LIN {X 0,Y 474.677,Z 139.36,A -85,B 0,C 180,E1 -7395.457,E2 -7395.457} C_VEL
LIN {X 0,Y 474.649,Z 139.359,A -85,B 0,C 180,E1 -7399.011,E2 -7399.011} C_VEL
LIN {X 0,Y 474.578,Z 139.368,A -85,B 0,C 180,E1 -7401.73,E2 -7401.73} C_VEL
LIN {X 0,Y 474.616,Z 139.361,A -85,B 0,C 180,E1 -7404.495,E2 -7404.495} C_VEL
LIN {X 0,Y 474.629,Z 139.365,A -85,B 0,C 180,E1 -7407.325,E2 -7407.325} C_VEL
LIN {X 0,Y 474.588,Z 139.364,A -85,B 0,C 180,E1 -7410.232,E2 -7410.232} C_VEL
LIN {X 0,Y 474.607,Z 139.367,A -85,B 0,C 180,E1 -7413.223,E2 -7413.223} C_VEL
LIN {X 0,Y 474.581,Z 139.366,A -85,B 0,C 180,E1 -7416.324,E2 -7416.324} C_VEL
LIN {X 0,Y 474.615,Z 139.361,A -85,B 0,C 180,E1 -7419.549,E2 -7419.549} C_VEL
LIN {X 0,Y 474.578,Z 139.367,A -85,B 0,C 180,E1 -7422.232,E2 -7422.232} C_VEL
LIN {X 0,Y 474.611,Z 139.362,A -85,B 0,C 180,E1 -7425.299,E2 -7425.299} C_VEL
LIN {X 0,Y 474.61,Z 139.364,A -85,B 0,C 180,E1 -7428.215,E2 -7428.215} C_VEL
LIN {X 0,Y 474.605,Z 139.362,A -85,B 0,C 180,E1 -7431.543,E2 -7431.543} C_VEL
LIN {X 0,Y 474.619,Z 139.364,A -85,B 0,C 180,E1 -7434.726,E2 -7434.726} C_VEL
LIN {X 0,Y 474.633,Z 139.36,A -85,B 0,C 180,E1 -7437.789,E2 -7437.789} C_VEL
LIN {X 0,Y 474.597,Z 139.364,A -85,B 0,C 180,E1 -7440.891,E2 -7440.891} C_VEL
LIN {X 0,Y 474.609,Z 139.363,A -85,B 0,C 180,E1 -7443.626,E2 -7443.626} C_VEL
LIN {X 0,Y 474.634,Z 139.36,A -85,B 0,C 180,E1 -7446.643,E2 -7446.643} C_VEL
LIN {X 0,Y 474.709,Z 139.506,A -85,B 0,C 180,E1 -7449.301,E2 -7449.301} C_VEL
LIN {X 0,Y 475.543,Z 144.063,A -85,B 0,C 180,E1 -7450.291,E2 -7450.291} C_VEL
LIN {X 0,Y 475.076,Z 146.121,A -85,B 0,C 180,E1 -7450.692,E2 -7450.692} C_VEL
LIN {X 0,Y 472.301,Z 149.701,A -85,B 0,C 180,E1 -7451.293,E2 -7451.293} C_VEL
LIN {X 0,Y 469.325,Z 153.345,A -85,B 0,C 180,E1 -7451.896,E2 -7451.896} C_VEL
LIN {X 0,Y 468.584,Z 155.513,A -85,B 0,C 180,E1 -7452.3,E2 -7452.3} C_VEL
LIN {X 0,Y 468.493,Z 159.191,A -85,B 0,C 180,E1 -7453.033,E2 -7453.033} C_VEL
LIN {X 0,Y 471.458,Z 174.816,A -85,B 0,C 180,E1 -7453.399,E2 -7453.399} C_VEL
LIN {X 0,Y 470.697,Z 266.818,A -85,B 0,C 180,E1 -7454.826,E2 -7454.826} C_VEL
LIN {X 0,Y 470.413,Z 279.928,A -85,B 0,C 180,E1 -7455.204,E2 -7455.204} C_VEL
LIN {X 0,Y 470.036,Z 291.987,A -85,B 0,C 180,E1 -7455.718,E2 -7455.718} C_VEL
LIN {X 0,Y 469.631,Z 303.292,A -85,B 0,C 180,E1 -7456.364,E2 -7456.364} C_VEL
LIN {X 0,Y 469.304,Z 313.727,A -85,B 0,C 180,E1 -7457.13,E2 -7457.13} C_VEL
LIN {X 0,Y 468.722,Z 324.409,A -85,B 0,C 180,E1 -7458.103,E2 -7458.103} C_VEL
LIN {X 0,Y 468.281,Z 334.015,A -85,B 0,C 180,E1 -7459.188,E2 -7459.188} C_VEL
LIN {X 0,Y 467.829,Z 341.883,A -85,B 0,C 180,E1 -7460.271,E2 -7460.271} C_VEL
LIN {X 0,Y 467.434,Z 349.574,A -85,B 0,C 180,E1 -7461.571,E2 -7461.571} C_VEL
LIN {X 0,Y 467.127,Z 356.625,A -85,B 0,C 180,E1 -7463.088,E2 -7463.088} C_VEL
LIN {X 0,Y 466.942,Z 361.324,A -85,B 0,C 180,E1 -7464.386,E2 -7464.386} C_VEL
LIN {X 0,Y 466.844,Z 364.92,A -85,B 0,C 180,E1 -7465.684,E2 -7465.684} C_VEL
LIN {X 0,Y 466.817,Z 366.778,A -85,B 0,C 180,E1 -7466.548,E2 -7466.548} C_VEL
LIN {X 0,Y 466.718,Z 368.181,A -85,B 0,C 180,E1 -7467.411,E2 -7467.411} C_VEL
LIN {X 0,Y 466.626,Z 369.793,A -85,B 0,C 180,E1 -7469.137,E2 -7469.137} C_VEL
LIN {X 0,Y 466.607,Z 370.029,A -85,B 0,C 180,E1 -7470,E2 -7470} C_VEL
LIN {X 0,Y 466.626,Z 369.843,A -85,B 0,C 180,E1 -7470.863,E2 -7470.863} C_VEL
LIN {X 0,Y 466.719,Z 368.296,A -85,B 0,C 180,E1 -7472.59,E2 -7472.59} C_VEL
LIN {X 0,Y 466.818,Z 366.942,A -85,B 0,C 180,E1 -7473.453,E2 -7473.453} C_VEL
LIN {X 0,Y 466.819,Z 364.087,A -85,B 0,C 180,E1 -7474.75,E2 -7474.75} C_VEL
LIN {X 0,Y 467.063,Z 360.207,A -85,B 0,C 180,E1 -7476.047,E2 -7476.047} C_VEL
LIN {X 0,Y 467.173,Z 355.208,A -85,B 0,C 180,E1 -7477.347,E2 -7477.347} C_VEL
LIN {X 0,Y 467.498,Z 348.91,A -85,B 0,C 180,E1 -7478.647,E2 -7478.647} C_VEL
LIN {X 0,Y 467.886,Z 341.024,A -85,B 0,C 180,E1 -7479.947,E2 -7479.947} C_VEL
LIN {X 0,Y 468.262,Z 332.985,A -85,B 0,C 180,E1 -7481.032,E2 -7481.032} C_VEL
LIN {X 0,Y 468.813,Z 323.168,A -85,B 0,C 180,E1 -7482.115,E2 -7482.115} C_VEL
LIN {X 0,Y 469.318,Z 312.035,A -85,B 0,C 180,E1 -7483.099,E2 -7483.099} C_VEL
LIN {X 0,Y 469.813,Z 299.55,A -85,B 0,C 180,E1 -7483.959,E2 -7483.959} C_VEL
LIN {X 0,Y 470.211,Z 288.228,A -85,B 0,C 180,E1 -7484.554,E2 -7484.554} C_VEL
LIN {X 0,Y 470.55,Z 275.334,A -85,B 0,C 180,E1 -7485.041,E2 -7485.041} C_VEL
LIN {X 0,Y 470.828,Z 261.566,A -85,B 0,C 180,E1 -7485.364,E2 -7485.364} C_VEL
LIN {X 0,Y 471.336,Z 173.724,A -85,B 0,C 180,E1 -7486.716,E2 -7486.716} C_VEL
LIN {X 0,Y 468.504,Z 159.186,A -85,B 0,C 180,E1 -7487.061,E2 -7487.061} C_VEL
LIN {X 0,Y 468.83,Z 147.183,A -85,B 0,C 180,E1 -7489.484,E2 -7489.484} C_VEL
LIN {X 0,Y 467.636,Z 140.236,A -85,B 0,C 180,E1 -7491.027,E2 -7491.027} C_VEL
LIN {X 0,Y 467.559,Z 140.247,A -85,B 0,C 180,E1 -7493.944,E2 -7493.944} C_VEL
LIN {X 0,Y 467.564,Z 140.239,A -85,B 0,C 180,E1 -7496.804,E2 -7496.804} C_VEL
LIN {X 0,Y 467.548,Z 140.248,A -85,B 0,C 180,E1 -7499.739,E2 -7499.739} C_VEL
LIN {X 0,Y 467.585,Z 140.236,A -85,B 0,C 180,E1 -7502.758,E2 -7502.758} C_VEL
LIN {X 0,Y 467.552,Z 140.245,A -85,B 0,C 180,E1 -7505.89,E2 -7505.89} C_VEL
LIN {X 0,Y 467.553,Z 140.243,A -85,B 0,C 180,E1 -7509.148,E2 -7509.148} C_VEL
LIN {X 0,Y 467.567,Z 140.246,A -85,B 0,C 180,E1 -7511.404,E2 -7511.404} C_VEL
LIN {X 0,Y 467.565,Z 140.241,A -85,B 0,C 180,E1 -7514.947,E2 -7514.947} C_VEL
LIN {X 0,Y 467.56,Z 140.245,A -85,B 0,C 180,E1 -7517.436,E2 -7517.436} C_VEL
LIN {X 0,Y 467.563,Z 140.239,A -85,B 0,C 180,E1 -7520.048,E2 -7520.048} C_VEL
LIN {X 0,Y 467.522,Z 140.251,A -85,B 0,C 180,E1 -7523.037,E2 -7523.037} C_VEL
LIN {X 0,Y 467.565,Z 140.239,A -85,B 0,C 180,E1 -7526.21,E2 -7526.21} C_VEL
LIN {X 0,Y 467.561,Z 140.243,A -85,B 0,C 180,E1 -7529.265,E2 -7529.265} C_VEL
LIN {X 0,Y 467.573,Z 140.241,A -85,B 0,C 180,E1 -7532.475,E2 -7532.475} C_VEL
LIN {X 0,Y 467.566,Z 140.242,A -85,B 0,C 180,E1 -7535.11,E2 -7535.11} C_VEL
LIN {X 0,Y 467.531,Z 140.243,A -85,B 0,C 180,E1 -7537.926,E2 -7537.926} C_VEL
LIN {X 0,Y 467.615,Z 140.24,A -85,B 0,C 180,E1 -7540.692,E2 -7540.692} C_VEL
LIN {X 0,Y 467.609,Z 140.238,A -85,B 0,C 180,E1 -7544.304,E2 -7544.304} C_VEL
LIN {X 0,Y 467.653,Z 140.229,A -85,B 0,C 180,E1 -7547.854,E2 -7547.854} C_VEL
LIN {X 0,Y 467.653,Z 140.228,A -85,B 0,C 180,E1 -7551.357,E2 -7551.357} C_VEL
LIN {X 0,Y 467.696,Z 140.227,A -85,B 0,C 180,E1 -7553.962,E2 -7553.962} C_VEL
LIN {X 0,Y 467.808,Z 140.209,A -85,B 0,C 180,E1 -7557.417,E2 -7557.417} C_VEL
LIN {X 0,Y 467.845,Z 140.211,A -85,B 0,C 180,E1 -7560,E2 -7560} C_VEL
LIN {X 0,Y 467.806,Z 140.21,A -85,B 0,C 180,E1 -7562.583,E2 -7562.583} C_VEL
LIN {X 0,Y 467.695,Z 140.229,A -85,B 0,C 180,E1 -7566.038,E2 -7566.038} C_VEL
LIN {X 0,Y 467.625,Z 140.231,A -85,B 0,C 180,E1 -7568.644,E2 -7568.644} C_VEL
LIN {X 0,Y 467.637,Z 140.232,A -85,B 0,C 180,E1 -7572.146,E2 -7572.146} C_VEL
LIN {X 0,Y 467.573,Z 140.245,A -85,B 0,C 180,E1 -7575.697,E2 -7575.697} C_VEL
LIN {X 0,Y 467.568,Z 140.238,A -85,B 0,C 180,E1 -7578.748,E2 -7578.748} C_VEL
LIN {X 0,Y 467.555,Z 140.245,A -85,B 0,C 180,E1 -7581.261,E2 -7581.261} C_VEL
LIN {X 0,Y 467.545,Z 140.243,A -85,B 0,C 180,E1 -7583.945,E2 -7583.945} C_VEL
LIN {X 0,Y 467.531,Z 140.245,A -85,B 0,C 180,E1 -7586.806,E2 -7586.806} C_VEL
LIN {X 0,Y 467.507,Z 140.248,A -85,B 0,C 180,E1 -7589.742,E2 -7589.742} C_VEL
LIN {X 0,Y 467.57,Z 140.241,A -85,B 0,C 180,E1 -7592.76,E2 -7592.76} C_VEL
LIN {X 0,Y 467.547,Z 140.241,A -85,B 0,C 180,E1 -7595.89,E2 -7595.89} C_VEL
LIN {X 0,Y 467.55,Z 140.246,A -85,B 0,C 180,E1 -7599.148,E2 -7599.148} C_VEL
LIN {X 0,Y 467.557,Z 140.242,A -85,B 0,C 180,E1 -7601.405,E2 -7601.405} C_VEL
LIN {X 0,Y 467.564,Z 140.243,A -85,B 0,C 180,E1 -7605.053,E2 -7605.053} C_VEL
LIN {X 0,Y 467.56,Z 140.247,A -85,B 0,C 180,E1 -7608.726,E2 -7608.726} C_VEL
LIN {X 0,Y 467.561,Z 140.24,A -85,B 0,C 180,E1 -7611.955,E2 -7611.955} C_VEL
LIN {X 0,Y 467.556,Z 140.241,A -85,B 0,C 180,E1 -7615.167,E2 -7615.167} C_VEL
LIN {X 0,Y 467.579,Z 140.243,A -85,B 0,C 180,E1 -7618.26,E2 -7618.26} C_VEL
LIN {X 0,Y 467.546,Z 140.244,A -85,B 0,C 180,E1 -7621.248,E2 -7621.248} C_VEL
LIN {X 0,Y 467.617,Z 140.444,A -85,B 0,C 180,E1 -7623.981,E2 -7623.981} C_VEL
LIN {X 0,Y 469.837,Z 152.033,A -85,B 0,C 180,E1 -7626.179,E2 -7626.179} C_VEL
LIN {X 0,Y 469.312,Z 165.507,A -85,B 0,C 180,E1 -7628.541,E2 -7628.541} C_VEL
LIN {X 0,Y 468.516,Z 184.729,A -85,B 0,C 180,E1 -7631.865,E2 -7631.865} C_VEL
LIN {X 0,Y 468.292,Z 191.201,A -85,B 0,C 180,E1 -7632.976,E2 -7632.976} C_VEL
LIN {X 0,Y 471.193,Z 211.474,A -85,B 0,C 180,E1 -7633.399,E2 -7633.399} C_VEL
LIN {X 0,Y 470.529,Z 299.617,A -85,B 0,C 180,E1 -7634.764,E2 -7634.764} C_VEL
LIN {X 0,Y 470.159,Z 312.891,A -85,B 0,C 180,E1 -7635.14,E2 -7635.14} C_VEL
LIN {X 0,Y 469.717,Z 325.06,A -85,B 0,C 180,E1 -7635.652,E2 -7635.652} C_VEL
LIN {X 0,Y 469.181,Z 337.34,A -85,B 0,C 180,E1 -7636.354,E2 -7636.354} C_VEL
LIN {X 0,Y 468.645,Z 349.413,A -85,B 0,C 180,E1 -7637.26,E2 -7637.26} C_VEL
LIN {X 0,Y 468.147,Z 360.453,A -85,B 0,C 180,E1 -7638.307,E2 -7638.307} C_VEL
LIN {X 0,Y 467.678,Z 369.639,A -85,B 0,C 180,E1 -7639.392,E2 -7639.392} C_VEL
LIN {X 0,Y 467.26,Z 378.592,A -85,B 0,C 180,E1 -7640.695,E2 -7640.695} C_VEL
LIN {X 0,Y 466.993,Z 385.802,A -85,B 0,C 180,E1 -7641.998,E2 -7641.998} C_VEL
LIN {X 0,Y 466.831,Z 390.669,A -85,B 0,C 180,E1 -7643.082,E2 -7643.082} C_VEL
LIN {X 0,Y 466.73,Z 395.401,A -85,B 0,C 180,E1 -7644.383,E2 -7644.383} C_VEL
LIN {X 0,Y 466.646,Z 399.016,A -85,B 0,C 180,E1 -7645.681,E2 -7645.681} C_VEL
LIN {X 0,Y 466.689,Z 400.884,A -85,B 0,C 180,E1 -7646.546,E2 -7646.546} C_VEL
LIN {X 0,Y 466.662,Z 402.283,A -85,B 0,C 180,E1 -7647.41,E2 -7647.41} C_VEL
LIN {X 0,Y 466.623,Z 403.889,A -85,B 0,C 180,E1 -7649.137,E2 -7649.137} C_VEL
LIN {X 0,Y 466.605,Z 404.106,A -85,B 0,C 180,E1 -7650,E2 -7650} C_VEL
LIN {X 0,Y 466.623,Z 403.89,A -85,B 0,C 180,E1 -7650.863,E2 -7650.863} C_VEL
LIN {X 0,Y 466.662,Z 402.285,A -85,B 0,C 180,E1 -7652.589,E2 -7652.589} C_VEL
LIN {X 0,Y 466.689,Z 400.887,A -85,B 0,C 180,E1 -7653.453,E2 -7653.453} C_VEL
LIN {X 0,Y 466.687,Z 397.944,A -85,B 0,C 180,E1 -7654.751,E2 -7654.751} C_VEL
LIN {X 0,Y 466.741,Z 393.962,A -85,B 0,C 180,E1 -7656.05,E2 -7656.05} C_VEL
LIN {X 0,Y 466.938,Z 387.841,A -85,B 0,C 180,E1 -7657.567,E2 -7657.567} C_VEL
LIN {X 0,Y 467.157,Z 381.152,A -85,B 0,C 180,E1 -7658.87,E2 -7658.87} C_VEL
LIN {X 0,Y 467.512,Z 372.856,A -85,B 0,C 180,E1 -7660.173,E2 -7660.173} C_VEL
LIN {X 0,Y 467.972,Z 364.359,A -85,B 0,C 180,E1 -7661.258,E2 -7661.258} C_VEL
LIN {X 0,Y 468.448,Z 354.322,A -85,B 0,C 180,E1 -7662.301,E2 -7662.301} C_VEL
LIN {X 0,Y 468.93,Z 343.472,A -85,B 0,C 180,E1 -7663.211,E2 -7663.211} C_VEL
LIN {X 0,Y 469.421,Z 332.089,A -85,B 0,C 180,E1 -7663.97,E2 -7663.97} C_VEL
LIN {X 0,Y 469.874,Z 320.415,A -85,B 0,C 180,E1 -7664.564,E2 -7664.564} C_VEL
LIN {X 0,Y 470.37,Z 306.969,A -85,B 0,C 180,E1 -7665.046,E2 -7665.046} C_VEL
LIN {X 0,Y 470.624,Z 293.68,A -85,B 0,C 180,E1 -7665.343,E2 -7665.343} C_VEL
LIN {X 0,Y 471.058,Z 209.349,A -85,B 0,C 180,E1 -7666.637,E2 -7666.637} C_VEL
LIN {X 0,Y 468.285,Z 191.129,A -85,B 0,C 180,E1 -7667.034,E2 -7667.034} C_VEL
LIN {X 0,Y 468.906,Z 174.273,A -85,B 0,C 180,E1 -7669.936,E2 -7669.936} C_VEL
LIN {X 0,Y 469.661,Z 157.261,A -85,B 0,C 180,E1 -7672.895,E2 -7672.895} C_VEL
LIN {X 0,Y 469.837,Z 152.015,A -85,B 0,C 180,E1 -7673.82,E2 -7673.82} C_VEL
LIN {X 0,Y 467.571,Z 140.245,A -85,B 0,C 180,E1 -7676.081,E2 -7676.081} C_VEL
LIN {X 0,Y 467.548,Z 140.247,A -85,B 0,C 180,E1 -7679.327,E2 -7679.327} C_VEL
LIN {X 0,Y 467.575,Z 140.243,A -85,B 0,C 180,E1 -7681.74,E2 -7681.74} C_VEL
LIN {X 0,Y 467.552,Z 140.241,A -85,B 0,C 180,E1 -7684.833,E2 -7684.833} C_VEL
LIN {X 0,Y 467.557,Z 140.241,A -85,B 0,C 180,E1 -7688.044,E2 -7688.044} C_VEL
LIN {X 0,Y 467.559,Z 140.246,A -85,B 0,C 180,E1 -7691.403,E2 -7691.403} C_VEL
LIN {X 0,Y 467.559,Z 140.245,A -85,B 0,C 180,E1 -7695.052,E2 -7695.052} C_VEL
LIN {X 0,Y 467.554,Z 140.243,A -85,B 0,C 180,E1 -7698.725,E2 -7698.725} C_VEL
LIN {X 0,Y 467.554,Z 140.24,A -85,B 0,C 180,E1 -7701.954,E2 -7701.954} C_VEL
LIN {X 0,Y 467.548,Z 140.246,A -85,B 0,C 180,E1 -7705.166,E2 -7705.166} C_VEL
LIN {X 0,Y 467.549,Z 140.242,A -85,B 0,C 180,E1 -7708.257,E2 -7708.257} C_VEL
LIN {X 0,Y 467.535,Z 140.245,A -85,B 0,C 180,E1 -7711.248,E2 -7711.248} C_VEL
LIN {X 0,Y 467.568,Z 140.243,A -85,B 0,C 180,E1 -7714.4,E2 -7714.4} C_VEL
LIN {X 0,Y 467.559,Z 140.242,A -85,B 0,C 180,E1 -7716.995,E2 -7716.995} C_VEL
LIN {X 0,Y 467.6,Z 140.235,A -85,B 0,C 180,E1 -7719.776,E2 -7719.776} C_VEL
LIN {X 0,Y 467.551,Z 140.248,A -85,B 0,C 180,E1 -7722.505,E2 -7722.505} C_VEL
LIN {X 0,Y 467.58,Z 140.237,A -85,B 0,C 180,E1 -7725.196,E2 -7725.196} C_VEL
LIN {X 0,Y 467.637,Z 140.232,A -85,B 0,C 180,E1 -7727.854,E2 -7727.854} C_VEL
LIN {X 0,Y 467.622,Z 140.232,A -85,B 0,C 180,E1 -7731.356,E2 -7731.356} C_VEL
LIN {X 0,Y 467.689,Z 140.229,A -85,B 0,C 180,E1 -7733.962,E2 -7733.962} C_VEL
LIN {X 0,Y 467.8,Z 140.21,A -85,B 0,C 180,E1 -7737.417,E2 -7737.417} C_VEL
LIN {X 0,Y 467.838,Z 140.212,A -85,B 0,C 180,E1 -7740,E2 -7740} C_VEL
LIN {X 0,Y 467.802,Z 140.21,A -85,B 0,C 180,E1 -7742.583,E2 -7742.583} C_VEL
LIN {X 0,Y 467.693,Z 140.227,A -85,B 0,C 180,E1 -7746.038,E2 -7746.038} C_VEL
LIN {X 0,Y 467.656,Z 140.227,A -85,B 0,C 180,E1 -7748.643,E2 -7748.643} C_VEL
LIN {X 0,Y 467.646,Z 140.23,A -85,B 0,C 180,E1 -7752.146,E2 -7752.146} C_VEL
LIN {X 0,Y 467.602,Z 140.24,A -85,B 0,C 180,E1 -7755.696,E2 -7755.696} C_VEL
LIN {X 0,Y 467.609,Z 140.24,A -85,B 0,C 180,E1 -7759.308,E2 -7759.308} C_VEL
LIN {X 0,Y 467.521,Z 140.245,A -85,B 0,C 180,E1 -7762.075,E2 -7762.075} C_VEL
LIN {X 0,Y 467.55,Z 140.244,A -85,B 0,C 180,E1 -7764.891,E2 -7764.891} C_VEL
LIN {X 0,Y 467.552,Z 140.242,A -85,B 0,C 180,E1 -7767.774,E2 -7767.774} C_VEL
LIN {X 0,Y 467.557,Z 140.247,A -85,B 0,C 180,E1 -7771.045,E2 -7771.045} C_VEL
LIN {X 0,Y 467.569,Z 140.238,A -85,B 0,C 180,E1 -7774.241,E2 -7774.241} C_VEL
LIN {X 0,Y 467.54,Z 140.246,A -85,B 0,C 180,E1 -7777.187,E2 -7777.187} C_VEL
LIN {X 0,Y 467.551,Z 140.242,A -85,B 0,C 180,E1 -7780.268,E2 -7780.268} C_VEL
LIN {X 0,Y 467.54,Z 140.242,A -85,B 0,C 180,E1 -7783.747,E2 -7783.747} C_VEL
LIN {X 0,Y 467.544,Z 140.244,A -85,B 0,C 180,E1 -7786.256,E2 -7786.256} C_VEL
LIN {X 0,Y 467.565,Z 140.239,A -85,B 0,C 180,E1 -7789.735,E2 -7789.735} C_VEL
LIN {X 0,Y 467.539,Z 140.246,A -85,B 0,C 180,E1 -7792.816,E2 -7792.816} C_VEL
LIN {X 0,Y 467.584,Z 140.242,A -85,B 0,C 180,E1 -7796.213,E2 -7796.213} C_VEL
LIN {X 0,Y 467.564,Z 140.239,A -85,B 0,C 180,E1 -7799.267,E2 -7799.267} C_VEL
LIN {X 0,Y 467.573,Z 140.242,A -85,B 0,C 180,E1 -7802.476,E2 -7802.476} C_VEL
LIN {X 0,Y 467.567,Z 140.238,A -85,B 0,C 180,E1 -7805.112,E2 -7805.112} C_VEL
LIN {X 0,Y 467.534,Z 140.249,A -85,B 0,C 180,E1 -7807.927,E2 -7807.927} C_VEL
LIN {X 0,Y 467.639,Z 140.342,A -85,B 0,C 180,E1 -7809.118,E2 -7809.118} C_VEL
LIN {X 0,Y 468.8,Z 146.733,A -85,B 0,C 180,E1 -7810.516,E2 -7810.516} C_VEL
LIN {X 0,Y 468.584,Z 155.513,A -85,B 0,C 180,E1 -7812.3,E2 -7812.3} C_VEL
LIN {X 0,Y 468.186,Z 157.697,A -85,B 0,C 180,E1 -7812.596,E2 -7812.596} C_VEL
LIN {X 0,Y 467.029,Z 161.3,A -85,B 0,C 180,E1 -7812.843,E2 -7812.843} C_VEL
LIN {X 0,Y 465.264,Z 166.866,A -85,B 0,C 180,E1 -7813.019,E2 -7813.019} C_VEL
LIN {X 0,Y 464.706,Z 170.912,A -85,B 0,C 180,E1 -7813.084,E2 -7813.084} C_VEL
LIN {X 0,Y 465.202,Z 178.355,A -85,B 0,C 180,E1 -7813.219,E2 -7813.219} C_VEL
LIN {X 0,Y 464.513,Z 185.835,A -85,B 0,C 180,E1 -7813.313,E2 -7813.313} C_VEL
LIN {X 0,Y 463.852,Z 267.095,A -85,B 0,C 180,E1 -7814.597,E2 -7814.597} C_VEL
LIN {X 0,Y 463.565,Z 280.958,A -85,B 0,C 180,E1 -7815.009,E2 -7815.009} C_VEL
LIN {X 0,Y 463.147,Z 293.361,A -85,B 0,C 180,E1 -7815.557,E2 -7815.557} C_VEL
LIN {X 0,Y 462.704,Z 305.342,A -85,B 0,C 180,E1 -7816.281,E2 -7816.281} C_VEL
LIN {X 0,Y 462.305,Z 316.561,A -85,B 0,C 180,E1 -7817.155,E2 -7817.155} C_VEL
LIN {X 0,Y 461.692,Z 326.795,A -85,B 0,C 180,E1 -7818.142,E2 -7818.142} C_VEL
LIN {X 0,Y 461.227,Z 335.973,A -85,B 0,C 180,E1 -7819.243,E2 -7819.243} C_VEL
LIN {X 0,Y 460.729,Z 344.88,A -85,B 0,C 180,E1 -7820.563,E2 -7820.563} C_VEL
LIN {X 0,Y 460.301,Z 352.051,A -85,B 0,C 180,E1 -7821.881,E2 -7821.881} C_VEL
LIN {X 0,Y 460.058,Z 357.769,A -85,B 0,C 180,E1 -7823.2,E2 -7823.2} C_VEL
LIN {X 0,Y 459.899,Z 361.583,A -85,B 0,C 180,E1 -7824.3,E2 -7824.3} C_VEL
LIN {X 0,Y 459.752,Z 365.181,A -85,B 0,C 180,E1 -7825.617,E2 -7825.617} C_VEL
LIN {X 0,Y 459.75,Z 367.037,A -85,B 0,C 180,E1 -7826.495,E2 -7826.495} C_VEL
LIN {X 0,Y 459.641,Z 368.441,A -85,B 0,C 180,E1 -7827.371,E2 -7827.371} C_VEL
LIN {X 0,Y 459.559,Z 370.052,A -85,B 0,C 180,E1 -7829.124,E2 -7829.124} C_VEL
LIN {X 0,Y 459.538,Z 370.287,A -85,B 0,C 180,E1 -7830,E2 -7830} C_VEL
LIN {X 0,Y 459.559,Z 370.101,A -85,B 0,C 180,E1 -7830.877,E2 -7830.877} C_VEL
LIN {X 0,Y 459.641,Z 368.554,A -85,B 0,C 180,E1 -7832.63,E2 -7832.63} C_VEL
LIN {X 0,Y 459.75,Z 367.199,A -85,B 0,C 180,E1 -7833.506,E2 -7833.506} C_VEL
LIN {X 0,Y 459.735,Z 364.345,A -85,B 0,C 180,E1 -7834.823,E2 -7834.823} C_VEL
LIN {X 0,Y 460.01,Z 360.464,A -85,B 0,C 180,E1 -7836.14,E2 -7836.14} C_VEL
LIN {X 0,Y 460.129,Z 355.465,A -85,B 0,C 180,E1 -7837.46,E2 -7837.46} C_VEL
LIN {X 0,Y 460.48,Z 349.167,A -85,B 0,C 180,E1 -7838.779,E2 -7838.779} C_VEL
LIN {X 0,Y 460.88,Z 341.281,A -85,B 0,C 180,E1 -7840.1,E2 -7840.1} C_VEL
LIN {X 0,Y 461.305,Z 333.24,A -85,B 0,C 180,E1 -7841.201,E2 -7841.201} C_VEL
LIN {X 0,Y 461.897,Z 323.422,A -85,B 0,C 180,E1 -7842.299,E2 -7842.299} C_VEL
LIN {X 0,Y 462.394,Z 312.863,A -85,B 0,C 180,E1 -7843.253,E2 -7843.253} C_VEL
LIN {X 0,Y 462.873,Z 301.561,A -85,B 0,C 180,E1 -7844.06,E2 -7844.06} C_VEL
LIN {X 0,Y 463.348,Z 289.604,A -85,B 0,C 180,E1 -7844.718,E2 -7844.718} C_VEL
LIN {X 0,Y 463.702,Z 276.492,A -85,B 0,C 180,E1 -7845.24,E2 -7845.24} C_VEL
LIN {X 0,Y 463.973,Z 263.305,A -85,B 0,C 180,E1 -7845.569,E2 -7845.569} C_VEL
LIN {X 0,Y 464.537,Z 174.717,A -85,B 0,C 180,E1 -7846.956,E2 -7846.956} C_VEL
LIN {X 0,Y 461.559,Z 159.464,A -85,B 0,C 180,E1 -7847.319,E2 -7847.319} C_VEL
LIN {X 0,Y 461.891,Z 148.48,A -85,B 0,C 180,E1 -7849.557,E2 -7849.557} C_VEL
LIN {X 0,Y 460.55,Z 141.119,A -85,B 0,C 180,E1 -7851.218,E2 -7851.218} C_VEL
LIN {X 0,Y 460.524,Z 141.12,A -85,B 0,C 180,E1 -7854.333,E2 -7854.333} C_VEL
LIN {X 0,Y 460.535,Z 141.115,A -85,B 0,C 180,E1 -7857.246,E2 -7857.246} C_VEL
LIN {X 0,Y 460.508,Z 141.12,A -85,B 0,C 180,E1 -7860.24,E2 -7860.24} C_VEL
LIN {X 0,Y 460.531,Z 141.118,A -85,B 0,C 180,E1 -7863.325,E2 -7863.325} C_VEL
LIN {X 0,Y 460.474,Z 141.122,A -85,B 0,C 180,E1 -7866.53,E2 -7866.53} C_VEL
LIN {X 0,Y 460.514,Z 141.12,A -85,B 0,C 180,E1 -7869.864,E2 -7869.864} C_VEL
LIN {X 0,Y 460.493,Z 141.121,A -85,B 0,C 180,E1 -7872.897,E2 -7872.897} C_VEL
LIN {X 0,Y 460.505,Z 141.12,A -85,B 0,C 180,E1 -7875.831,E2 -7875.831} C_VEL
LIN {X 0,Y 460.519,Z 141.121,A -85,B 0,C 180,E1 -7878.987,E2 -7878.987} C_VEL
LIN {X 0,Y 460.513,Z 141.124,A -85,B 0,C 180,E1 -7881.265,E2 -7881.265} C_VEL
LIN {X 0,Y 460.505,Z 141.12,A -85,B 0,C 180,E1 -7884.554,E2 -7884.554} C_VEL
LIN {X 0,Y 460.516,Z 141.117,A -85,B 0,C 180,E1 -7887.714,E2 -7887.714} C_VEL
LIN {X 0,Y 460.518,Z 141.123,A -85,B 0,C 180,E1 -7890.767,E2 -7890.767} C_VEL
LIN {X 0,Y 460.527,Z 141.115,A -85,B 0,C 180,E1 -7893.732,E2 -7893.732} C_VEL
LIN {X 0,Y 460.541,Z 141.12,A -85,B 0,C 180,E1 -7896.624,E2 -7896.624} C_VEL
LIN {X 0,Y 460.546,Z 141.113,A -85,B 0,C 180,E1 -7899.452,E2 -7899.452} C_VEL
LIN {X 0,Y 460.521,Z 141.119,A -85,B 0,C 180,E1 -7902.229,E2 -7902.229} C_VEL
LIN {X 0,Y 460.545,Z 141.116,A -85,B 0,C 180,E1 -7904.964,E2 -7904.964} C_VEL
LIN {X 0,Y 460.605,Z 141.111,A -85,B 0,C 180,E1 -7908.559,E2 -7908.559} C_VEL
LIN {X 0,Y 460.605,Z 141.106,A -85,B 0,C 180,E1 -7911.223,E2 -7911.223} C_VEL
LIN {X 0,Y 460.662,Z 141.102,A -85,B 0,C 180,E1 -7913.869,E2 -7913.869} C_VEL
LIN {X 0,Y 460.752,Z 141.088,A -85,B 0,C 180,E1 -7917.377,E2 -7917.377} C_VEL
LIN {X 0,Y 460.814,Z 141.087,A -85,B 0,C 180,E1 -7920,E2 -7920} C_VEL
LIN {X 0,Y 460.75,Z 141.089,A -85,B 0,C 180,E1 -7922.623,E2 -7922.623} C_VEL
LIN {X 0,Y 460.661,Z 141.104,A -85,B 0,C 180,E1 -7926.131,E2 -7926.131} C_VEL
LIN {X 0,Y 460.58,Z 141.109,A -85,B 0,C 180,E1 -7928.777,E2 -7928.777} C_VEL
LIN {X 0,Y 460.594,Z 141.108,A -85,B 0,C 180,E1 -7932.435,E2 -7932.435} C_VEL
LIN {X 0,Y 460.522,Z 141.119,A -85,B 0,C 180,E1 -7935.965,E2 -7935.965} C_VEL
LIN {X 0,Y 460.527,Z 141.116,A -85,B 0,C 180,E1 -7938.886,E2 -7938.886} C_VEL
LIN {X 0,Y 460.506,Z 141.126,A -85,B 0,C 180,E1 -7941.486,E2 -7941.486} C_VEL
LIN {X 0,Y 460.51,Z 141.117,A -85,B 0,C 180,E1 -7944.334,E2 -7944.334} C_VEL
LIN {X 0,Y 460.486,Z 141.128,A -85,B 0,C 180,E1 -7947.249,E2 -7947.249} C_VEL
LIN {X 0,Y 460.476,Z 141.122,A -85,B 0,C 180,E1 -7950.243,E2 -7950.243} C_VEL
LIN {X 0,Y 460.513,Z 141.122,A -85,B 0,C 180,E1 -7953.326,E2 -7953.326} C_VEL
LIN {X 0,Y 460.469,Z 141.125,A -85,B 0,C 180,E1 -7956.53,E2 -7956.53} C_VEL
LIN {X 0,Y 460.511,Z 141.117,A -85,B 0,C 180,E1 -7959.865,E2 -7959.865} C_VEL
LIN {X 0,Y 460.461,Z 141.131,A -85,B 0,C 180,E1 -7962.894,E2 -7962.894} C_VEL
LIN {X 0,Y 460.502,Z 141.118,A -85,B 0,C 180,E1 -7965.832,E2 -7965.832} C_VEL
LIN {X 0,Y 460.514,Z 141.121,A -85,B 0,C 180,E1 -7968.987,E2 -7968.987} C_VEL
LIN {X 0,Y 460.498,Z 141.124,A -85,B 0,C 180,E1 -7972.377,E2 -7972.377} C_VEL
LIN {X 0,Y 460.536,Z 141.114,A -85,B 0,C 180,E1 -7975.623,E2 -7975.623} C_VEL
LIN {X 0,Y 460.539,Z 141.119,A -85,B 0,C 180,E1 -7978.745,E2 -7978.745} C_VEL
LIN {X 0,Y 460.533,Z 141.122,A -85,B 0,C 180,E1 -7982.266,E2 -7982.266} C_VEL
LIN {X 0,Y 460.525,Z 141.165,A -85,B 0,C 180,E1 -7983.732,E2 -7983.732} C_VEL
LIN {X 0,Y 462.868,Z 153.087,A -85,B 0,C 180,E1 -7986.036,E2 -7986.036} C_VEL
LIN {X 0,Y 462.408,Z 165.676,A -85,B 0,C 180,E1 -7988.281,E2 -7988.281} C_VEL
LIN {X 0,Y 461.542,Z 184.468,A -85,B 0,C 180,E1 -7991.581,E2 -7991.581} C_VEL
LIN {X 0,Y 461.3,Z 190.939,A -85,B 0,C 180,E1 -7992.709,E2 -7992.709} C_VEL
LIN {X 0,Y 464.372,Z 212.253,A -85,B 0,C 180,E1 -7993.164,E2 -7993.164} C_VEL
LIN {X 0,Y 463.686,Z 299.369,A -85,B 0,C 180,E1 -7994.534,E2 -7994.534} C_VEL
LIN {X 0,Y 463.3,Z 312.639,A -85,B 0,C 180,E1 -7994.915,E2 -7994.915} C_VEL
LIN {X 0,Y 462.813,Z 324.805,A -85,B 0,C 180,E1 -7995.433,E2 -7995.433} C_VEL
LIN {X 0,Y 462.259,Z 337.084,A -85,B 0,C 180,E1 -7996.145,E2 -7996.145} C_VEL
LIN {X 0,Y 461.706,Z 349.156,A -85,B 0,C 180,E1 -7997.065,E2 -7997.065} C_VEL
LIN {X 0,Y 461.169,Z 360.196,A -85,B 0,C 180,E1 -7998.127,E2 -7998.127} C_VEL
LIN {X 0,Y 460.644,Z 369.379,A -85,B 0,C 180,E1 -7999.228,E2 -7999.228} C_VEL
LIN {X 0,Y 460.212,Z 378.333,A -85,B 0,C 180,E1 -8000.551,E2 -8000.551} C_VEL
LIN {X 0,Y 459.92,Z 385.542,A -85,B 0,C 180,E1 -8001.874,E2 -8001.874} C_VEL
LIN {X 0,Y 459.745,Z 390.409,A -85,B 0,C 180,E1 -8002.975,E2 -8002.975} C_VEL
LIN {X 0,Y 459.629,Z 395.142,A -85,B 0,C 180,E1 -8004.296,E2 -8004.296} C_VEL
LIN {X 0,Y 459.563,Z 398.758,A -85,B 0,C 180,E1 -8005.614,E2 -8005.614} C_VEL
LIN {X 0,Y 459.585,Z 400.625,A -85,B 0,C 180,E1 -8006.493,E2 -8006.493} C_VEL
LIN {X 0,Y 459.584,Z 402.024,A -85,B 0,C 180,E1 -8007.37,E2 -8007.37} C_VEL
LIN {X 0,Y 459.555,Z 403.631,A -85,B 0,C 180,E1 -8009.123,E2 -8009.123} C_VEL
LIN {X 0,Y 459.536,Z 403.848,A -85,B 0,C 180,E1 -8010,E2 -8010} C_VEL
LIN {X 0,Y 459.555,Z 403.631,A -85,B 0,C 180,E1 -8010.876,E2 -8010.876} C_VEL
LIN {X 0,Y 459.584,Z 402.026,A -85,B 0,C 180,E1 -8012.629,E2 -8012.629} C_VEL
LIN {X 0,Y 459.584,Z 400.627,A -85,B 0,C 180,E1 -8013.506,E2 -8013.506} C_VEL
LIN {X 0,Y 459.614,Z 397.684,A -85,B 0,C 180,E1 -8014.824,E2 -8014.824} C_VEL
LIN {X 0,Y 459.714,Z 392.67,A -85,B 0,C 180,E1 -8016.43,E2 -8016.43} C_VEL
LIN {X 0,Y 459.881,Z 386.564,A -85,B 0,C 180,E1 -8017.905,E2 -8017.905} C_VEL
LIN {X 0,Y 460.167,Z 379.651,A -85,B 0,C 180,E1 -8019.227,E2 -8019.227} C_VEL
LIN {X 0,Y 460.468,Z 372.593,A -85,B 0,C 180,E1 -8020.331,E2 -8020.331} C_VEL
LIN {X 0,Y 460.976,Z 364.096,A -85,B 0,C 180,E1 -8021.431,E2 -8021.431} C_VEL
LIN {X 0,Y 461.474,Z 354.273,A -85,B 0,C 180,E1 -8022.469,E2 -8022.469} C_VEL
LIN {X 0,Y 462.004,Z 343.208,A -85,B 0,C 180,E1 -8023.413,E2 -8023.413} C_VEL
LIN {X 0,Y 462.512,Z 331.824,A -85,B 0,C 180,E1 -8024.183,E2 -8024.183} C_VEL
LIN {X 0,Y 463.011,Z 320.15,A -85,B 0,C 180,E1 -8024.784,E2 -8024.784} C_VEL
LIN {X 0,Y 463.454,Z 307.615,A -85,B 0,C 180,E1 -8025.248,E2 -8025.248} C_VEL
LIN {X 0,Y 463.773,Z 294.925,A -85,B 0,C 180,E1 -8025.547,E2 -8025.547} C_VEL
LIN {X 0,Y 464.291,Z 210.428,A -85,B 0,C 180,E1 -8026.865,E2 -8026.865} C_VEL
LIN {X 0,Y 461.322,Z 190.929,A -85,B 0,C 180,E1 -8027.288,E2 -8027.288} C_VEL
LIN {X 0,Y 461.996,Z 174.012,A -85,B 0,C 180,E1 -8030.247,E2 -8030.247} C_VEL
LIN {X 0,Y 462.791,Z 157.002,A -85,B 0,C 180,E1 -8033.255,E2 -8033.255} C_VEL
LIN {X 0,Y 462.877,Z 153.065,A -85,B 0,C 180,E1 -8033.963,E2 -8033.963} C_VEL
LIN {X 0,Y 460.534,Z 141.121,A -85,B 0,C 180,E1 -8036.297,E2 -8036.297} C_VEL
LIN {X 0,Y 460.514,Z 141.124,A -85,B 0,C 180,E1 -8039.554,E2 -8039.554} C_VEL
LIN {X 0,Y 460.522,Z 141.117,A -85,B 0,C 180,E1 -8042.284,E2 -8042.284} C_VEL
LIN {X 0,Y 460.502,Z 141.126,A -85,B 0,C 180,E1 -8045.445,E2 -8045.445} C_VEL
LIN {X 0,Y 460.499,Z 141.121,A -85,B 0,C 180,E1 -8048.89,E2 -8048.89} C_VEL
LIN {X 0,Y 460.504,Z 141.122,A -85,B 0,C 180,E1 -8051.598,E2 -8051.598} C_VEL
LIN {X 0,Y 460.506,Z 141.119,A -85,B 0,C 180,E1 -8054.588,E2 -8054.588} C_VEL
LIN {X 0,Y 460.472,Z 141.123,A -85,B 0,C 180,E1 -8057.813,E2 -8057.813} C_VEL
LIN {X 0,Y 460.505,Z 141.118,A -85,B 0,C 180,E1 -8060.135,E2 -8060.135} C_VEL
LIN {X 0,Y 460.465,Z 141.125,A -85,B 0,C 180,E1 -8063.469,E2 -8063.469} C_VEL
LIN {X 0,Y 460.508,Z 141.123,A -85,B 0,C 180,E1 -8066.673,E2 -8066.673} C_VEL
LIN {X 0,Y 460.493,Z 141.12,A -85,B 0,C 180,E1 -8069.759,E2 -8069.759} C_VEL
LIN {X 0,Y 460.483,Z 141.129,A -85,B 0,C 180,E1 -8072.75,E2 -8072.75} C_VEL
LIN {X 0,Y 460.508,Z 141.118,A -85,B 0,C 180,E1 -8075.666,E2 -8075.666} C_VEL
LIN {X 0,Y 460.509,Z 141.126,A -85,B 0,C 180,E1 -8078.579,E2 -8078.579} C_VEL
LIN {X 0,Y 460.571,Z 141.11,A -85,B 0,C 180,E1 -8081.31,E2 -8081.31} C_VEL
LIN {X 0,Y 460.537,Z 141.116,A -85,B 0,C 180,E1 -8084.964,E2 -8084.964} C_VEL
LIN {X 0,Y 460.581,Z 141.113,A -85,B 0,C 180,E1 -8088.559,E2 -8088.559} C_VEL
LIN {X 0,Y 460.612,Z 141.112,A -85,B 0,C 180,E1 -8092.107,E2 -8092.107} C_VEL
LIN {X 0,Y 460.661,Z 141.1,A -85,B 0,C 180,E1 -8094.748,E2 -8094.748} C_VEL
LIN {X 0,Y 460.744,Z 141.089,A -85,B 0,C 180,E1 -8097.377,E2 -8097.377} C_VEL
LIN {X 0,Y 460.808,Z 141.088,A -85,B 0,C 180,E1 -8100,E2 -8100} C_VEL
LIN {X 0,Y 460.745,Z 141.089,A -85,B 0,C 180,E1 -8102.623,E2 -8102.623} C_VEL
LIN {X 0,Y 460.66,Z 141.102,A -85,B 0,C 180,E1 -8106.131,E2 -8106.131} C_VEL
LIN {X 0,Y 460.606,Z 141.105,A -85,B 0,C 180,E1 -8108.777,E2 -8108.777} C_VEL
LIN {X 0,Y 460.587,Z 141.108,A -85,B 0,C 180,E1 -8112.435,E2 -8112.435} C_VEL
LIN {X 0,Y 460.547,Z 141.115,A -85,B 0,C 180,E1 -8115.979,E2 -8115.979} C_VEL
LIN {X 0,Y 460.556,Z 141.117,A -85,B 0,C 180,E1 -8119.616,E2 -8119.616} C_VEL
LIN {X 0,Y 460.498,Z 141.119,A -85,B 0,C 180,E1 -8122.429,E2 -8122.429} C_VEL
LIN {X 0,Y 460.526,Z 141.117,A -85,B 0,C 180,E1 -8125.794,E2 -8125.794} C_VEL
LIN {X 0,Y 460.505,Z 141.118,A -85,B 0,C 180,E1 -8128.236,E2 -8128.236} C_VEL
LIN {X 0,Y 460.512,Z 141.123,A -85,B 0,C 180,E1 -8131.283,E2 -8131.283} C_VEL
LIN {X 0,Y 460.515,Z 141.119,A -85,B 0,C 180,E1 -8134.505,E2 -8134.505} C_VEL
LIN {X 0,Y 460.494,Z 141.12,A -85,B 0,C 180,E1 -8137.624,E2 -8137.624} C_VEL
LIN {X 0,Y 460.517,Z 141.118,A -85,B 0,C 180,E1 -8140.268,E2 -8140.268} C_VEL
LIN {X 0,Y 460.497,Z 141.12,A -85,B 0,C 180,E1 -8143.376,E2 -8143.376} C_VEL
LIN {X 0,Y 460.504,Z 141.126,A -85,B 0,C 180,E1 -8146.627,E2 -8146.627} C_VEL
LIN {X 0,Y 460.53,Z 141.115,A -85,B 0,C 180,E1 -8149.733,E2 -8149.733} C_VEL
LIN {X 0,Y 460.493,Z 141.127,A -85,B 0,C 180,E1 -8152.525,E2 -8152.525} C_VEL
LIN {X 0,Y 460.543,Z 141.114,A -85,B 0,C 180,E1 -8155.625,E2 -8155.625} C_VEL
LIN {X 0,Y 460.536,Z 141.117,A -85,B 0,C 180,E1 -8158.745,E2 -8158.745} C_VEL
LIN {X 0,Y 460.537,Z 141.122,A -85,B 0,C 180,E1 -8162.265,E2 -8162.265} C_VEL
LIN {X 0,Y 460.533,Z 141.116,A -85,B 0,C 180,E1 -8164.705,E2 -8164.705} C_VEL
LIN {X 0,Y 460.51,Z 141.12,A -85,B 0,C 180,E1 -8167.572,E2 -8167.572} C_VEL
LIN {X 0,Y 460.591,Z 141.24,A -85,B 0,C 180,E1 -8168.937,E2 -8168.937} C_VEL
LIN {X 0,Y 461.84,Z 148.03,A -85,B 0,C 180,E1 -8170.441,E2 -8170.441} C_VEL
LIN {X 0,Y 461.548,Z 159.423,A -85,B 0,C 180,E1 -8172.767,E2 -8172.767} C_VEL
LIN {X 0,Y 464.656,Z 175.108,A -85,B 0,C 180,E1 -8173.148,E2 -8173.148} C_VEL
LIN {X 0,Y 464.513,Z 185.835,A -85,B 0,C 180,E1 -8173.313,E2 -8173.313} C_VEL
LIN {X 0,Y 463.84,Z 191.681,A -85,B 0,C 180,E1 -8173.38,E2 -8173.38} C_VEL
LIN {X 0,Y 458.223,Z 210.695,A -85,B 0,C 180,E1 -8173.472,E2 -8173.472} C_VEL
LIN {X 0,Y 457.574,Z 216.54,A -85,B 0,C 180,E1 -8173.541,E2 -8173.541} C_VEL
LIN {X 0,Y 457.02,Z 267.371,A -85,B 0,C 180,E1 -8174.361,E2 -8174.361} C_VEL
LIN {X 0,Y 456.741,Z 281.228,A -85,B 0,C 180,E1 -8174.78,E2 -8174.78} C_VEL
LIN {X 0,Y 456.283,Z 293.628,A -85,B 0,C 180,E1 -8175.335,E2 -8175.335} C_VEL
LIN {X 0,Y 455.806,Z 305.91,A -85,B 0,C 180,E1 -8176.091,E2 -8176.091} C_VEL
LIN {X 0,Y 455.394,Z 316.825,A -85,B 0,C 180,E1 -8176.956,E2 -8176.956} C_VEL
LIN {X 0,Y 454.748,Z 327.059,A -85,B 0,C 180,E1 -8177.958,E2 -8177.958} C_VEL
LIN {X 0,Y 454.264,Z 336.234,A -85,B 0,C 180,E1 -8179.076,E2 -8179.076} C_VEL
LIN {X 0,Y 453.732,Z 345.142,A -85,B 0,C 180,E1 -8180.416,E2 -8180.416} C_VEL
LIN {X 0,Y 453.282,Z 352.313,A -85,B 0,C 180,E1 -8181.755,E2 -8181.755} C_VEL
LIN {X 0,Y 452.994,Z 358.365,A -85,B 0,C 180,E1 -8183.186,E2 -8183.186} C_VEL
LIN {X 0,Y 452.722,Z 363.159,A -85,B 0,C 180,E1 -8184.656,E2 -8184.656} C_VEL
LIN {X 0,Y 452.661,Z 365.441,A -85,B 0,C 180,E1 -8185.548,E2 -8185.548} C_VEL
LIN {X 0,Y 452.684,Z 367.297,A -85,B 0,C 180,E1 -8186.44,E2 -8186.44} C_VEL
LIN {X 0,Y 452.567,Z 368.7,A -85,B 0,C 180,E1 -8187.33,E2 -8187.33} C_VEL
LIN {X 0,Y 452.464,Z 370.311,A -85,B 0,C 180,E1 -8189.11,E2 -8189.11} C_VEL
LIN {X 0,Y 452.472,Z 370.545,A -85,B 0,C 180,E1 -8190,E2 -8190} C_VEL
LIN {X 0,Y 452.464,Z 370.36,A -85,B 0,C 180,E1 -8190.89,E2 -8190.89} C_VEL
LIN {X 0,Y 452.567,Z 368.812,A -85,B 0,C 180,E1 -8192.671,E2 -8192.671} C_VEL
LIN {X 0,Y 452.684,Z 367.457,A -85,B 0,C 180,E1 -8193.561,E2 -8193.561} C_VEL
LIN {X 0,Y 452.659,Z 364.603,A -85,B 0,C 180,E1 -8194.899,E2 -8194.899} C_VEL
LIN {X 0,Y 452.957,Z 360.722,A -85,B 0,C 180,E1 -8196.236,E2 -8196.236} C_VEL
LIN {X 0,Y 453.081,Z 355.723,A -85,B 0,C 180,E1 -8197.577,E2 -8197.577} C_VEL
LIN {X 0,Y 453.451,Z 349.424,A -85,B 0,C 180,E1 -8198.917,E2 -8198.917} C_VEL
LIN {X 0,Y 453.884,Z 341.537,A -85,B 0,C 180,E1 -8200.258,E2 -8200.258} C_VEL
LIN {X 0,Y 454.33,Z 333.496,A -85,B 0,C 180,E1 -8201.375,E2 -8201.375} C_VEL
LIN {X 0,Y 454.971,Z 323.676,A -85,B 0,C 180,E1 -8202.49,E2 -8202.49} C_VEL
LIN {X 0,Y 455.503,Z 312.525,A -85,B 0,C 180,E1 -8203.505,E2 -8203.505} C_VEL
LIN {X 0,Y 456.081,Z 300.053,A -85,B 0,C 180,E1 -8204.388,E2 -8204.388} C_VEL
LIN {X 0,Y 456.501,Z 288.728,A -85,B 0,C 180,E1 -8205.001,E2 -8205.001} C_VEL
LIN {X 0,Y 456.893,Z 275.822,A -85,B 0,C 180,E1 -8205.502,E2 -8205.502} C_VEL
LIN {X 0,Y 457.18,Z 262.037,A -85,B 0,C 180,E1 -8205.835,E2 -8205.835} C_VEL
LIN {X 0,Y 457.763,Z 175.65,A -85,B 0,C 180,E1 -8207.203,E2 -8207.203} C_VEL
LIN {X 0,Y 454.616,Z 159.708,A -85,B 0,C 180,E1 -8207.592,E2 -8207.592} C_VEL
LIN {X 0,Y 454.938,Z 150.191,A -85,B 0,C 180,E1 -8209.55,E2 -8209.55} C_VEL
LIN {X 0,Y 453.587,Z 142.457,A -85,B 0,C 180,E1 -8211.27,E2 -8211.27} C_VEL
LIN {X 0,Y 453.504,Z 141.997,A -85,B 0,C 180,E1 -8211.375,E2 -8211.375} C_VEL
LIN {X 0,Y 453.496,Z 141.993,A -85,B 0,C 180,E1 -8214.736,E2 -8214.736} C_VEL
LIN {X 0,Y 453.508,Z 141.996,A -85,B 0,C 180,E1 -8217.953,E2 -8217.953} C_VEL
LIN {X 0,Y 453.477,Z 141.994,A -85,B 0,C 180,E1 -8220.759,E2 -8220.759} C_VEL
LIN {X 0,Y 453.478,Z 141.998,A -85,B 0,C 180,E1 -8223.913,E2 -8223.913} C_VEL
LIN {X 0,Y 453.45,Z 142,A -85,B 0,C 180,E1 -8227.19,E2 -8227.19} C_VEL
LIN {X 0,Y 453.471,Z 141.994,A -85,B 0,C 180,E1 -8230.611,E2 -8230.611} C_VEL
LIN {X 0,Y 453.46,Z 141.996,A -85,B 0,C 180,E1 -8234.222,E2 -8234.222} C_VEL
LIN {X 0,Y 453.448,Z 142.001,A -85,B 0,C 180,E1 -8237.003,E2 -8237.003} C_VEL
LIN {X 0,Y 453.47,Z 142,A -85,B 0,C 180,E1 -8239.412,E2 -8239.412} C_VEL
LIN {X 0,Y 453.448,Z 142.001,A -85,B 0,C 180,E1 -8242.81,E2 -8242.81} C_VEL
LIN {X 0,Y 453.465,Z 141.995,A -85,B 0,C 180,E1 -8246.086,E2 -8246.086} C_VEL
LIN {X 0,Y 453.463,Z 141.999,A -85,B 0,C 180,E1 -8249.239,E2 -8249.239} C_VEL
LIN {X 0,Y 453.488,Z 141.994,A -85,B 0,C 180,E1 -8252.294,E2 -8252.294} C_VEL
LIN {X 0,Y 453.491,Z 141.994,A -85,B 0,C 180,E1 -8255.264,E2 -8255.264} C_VEL
LIN {X 0,Y 453.478,Z 141.998,A -85,B 0,C 180,E1 -8258.415,E2 -8258.415} C_VEL
LIN {X 0,Y 453.52,Z 141.991,A -85,B 0,C 180,E1 -8261.008,E2 -8261.008} C_VEL
LIN {X 0,Y 453.515,Z 141.994,A -85,B 0,C 180,E1 -8264.725,E2 -8264.725} C_VEL
LIN {X 0,Y 453.555,Z 141.992,A -85,B 0,C 180,E1 -8268.379,E2 -8268.379} C_VEL
LIN {X 0,Y 453.573,Z 141.982,A -85,B 0,C 180,E1 -8271.086,E2 -8271.086} C_VEL
LIN {X 0,Y 453.63,Z 141.977,A -85,B 0,C 180,E1 -8273.774,E2 -8273.774} C_VEL
LIN {X 0,Y 453.698,Z 141.966,A -85,B 0,C 180,E1 -8277.336,E2 -8277.336} C_VEL
LIN {X 0,Y 453.763,Z 141.965,A -85,B 0,C 180,E1 -8280,E2 -8280} C_VEL
LIN {X 0,Y 453.697,Z 141.967,A -85,B 0,C 180,E1 -8282.664,E2 -8282.664} C_VEL
LIN {X 0,Y 453.629,Z 141.978,A -85,B 0,C 180,E1 -8286.226,E2 -8286.226} C_VEL
LIN {X 0,Y 453.551,Z 141.984,A -85,B 0,C 180,E1 -8288.914,E2 -8288.914} C_VEL
LIN {X 0,Y 453.562,Z 141.983,A -85,B 0,C 180,E1 -8292.529,E2 -8292.529} C_VEL
LIN {X 0,Y 453.482,Z 141.994,A -85,B 0,C 180,E1 -8296.198,E2 -8296.198} C_VEL
LIN {X 0,Y 453.482,Z 141.995,A -85,B 0,C 180,E1 -8299.028,E2 -8299.028} C_VEL
LIN {X 0,Y 453.466,Z 141.998,A -85,B 0,C 180,E1 -8301.837,E2 -8301.837} C_VEL
LIN {X 0,Y 453.464,Z 141.996,A -85,B 0,C 180,E1 -8304.737,E2 -8304.737} C_VEL
LIN {X 0,Y 453.454,Z 141.997,A -85,B 0,C 180,E1 -8307.941,E2 -8307.941} C_VEL
LIN {X 0,Y 453.444,Z 142,A -85,B 0,C 180,E1 -8310.762,E2 -8310.762} C_VEL
LIN {X 0,Y 453.464,Z 141.996,A -85,B 0,C 180,E1 -8313.914,E2 -8313.914} C_VEL
LIN {X 0,Y 453.447,Z 142.003,A -85,B 0,C 180,E1 -8317.19,E2 -8317.19} C_VEL
LIN {X 0,Y 453.469,Z 141.999,A -85,B 0,C 180,E1 -8320.612,E2 -8320.612} C_VEL
LIN {X 0,Y 453.48,Z 141.997,A -85,B 0,C 180,E1 -8324.529,E2 -8324.529} C_VEL
LIN {X 0,Y 453.435,Z 142,A -85,B 0,C 180,E1 -8328.071,E2 -8328.071} C_VEL
LIN {X 0,Y 453.448,Z 142.003,A -85,B 0,C 180,E1 -8330.801,E2 -8330.801} C_VEL
LIN {X 0,Y 453.451,Z 141.998,A -85,B 0,C 180,E1 -8333.917,E2 -8333.917} C_VEL
LIN {X 0,Y 453.475,Z 141.995,A -85,B 0,C 180,E1 -8337.151,E2 -8337.151} C_VEL
LIN {X 0,Y 453.464,Z 142.003,A -85,B 0,C 180,E1 -8340.267,E2 -8340.267} C_VEL
LIN {X 0,Y 453.509,Z 142.113,A -85,B 0,C 180,E1 -8343.523,E2 -8343.523} C_VEL
LIN {X 0,Y 455.913,Z 154.345,A -85,B 0,C 180,E1 -8345.927,E2 -8345.927} C_VEL
LIN {X 0,Y 455.546,Z 165.195,A -85,B 0,C 180,E1 -8347.896,E2 -8347.896} C_VEL
LIN {X 0,Y 454.616,Z 184.208,A -85,B 0,C 180,E1 -8351.29,E2 -8351.29} C_VEL
LIN {X 0,Y 454.348,Z 190.656,A -85,B 0,C 180,E1 -8352.433,E2 -8352.433} C_VEL
LIN {X 0,Y 457.584,Z 212.012,A -85,B 0,C 180,E1 -8352.906,E2 -8352.906} C_VEL
LIN {X 0,Y 456.854,Z 299.122,A -85,B 0,C 180,E1 -8354.297,E2 -8354.297} C_VEL
LIN {X 0,Y 456.454,Z 312.388,A -85,B 0,C 180,E1 -8354.683,E2 -8354.683} C_VEL
LIN {X 0,Y 455.89,Z 325.673,A -85,B 0,C 180,E1 -8355.264,E2 -8355.264} C_VEL
LIN {X 0,Y 455.349,Z 336.828,A -85,B 0,C 180,E1 -8355.931,E2 -8355.931} C_VEL
LIN {X 0,Y 454.764,Z 348.278,A -85,B 0,C 180,E1 -8356.81,E2 -8356.81} C_VEL
LIN {X 0,Y 454.274,Z 358.893,A -85,B 0,C 180,E1 -8357.831,E2 -8357.831} C_VEL
LIN {X 0,Y 453.77,Z 367.441,A -85,B 0,C 180,E1 -8358.837,E2 -8358.837} C_VEL
LIN {X 0,Y 453.333,Z 375.331,A -85,B 0,C 180,E1 -8359.955,E2 -8359.955} C_VEL
LIN {X 0,Y 452.982,Z 383.041,A -85,B 0,C 180,E1 -8361.299,E2 -8361.299} C_VEL
LIN {X 0,Y 452.674,Z 390.15,A -85,B 0,C 180,E1 -8362.865,E2 -8362.865} C_VEL
LIN {X 0,Y 452.531,Z 394.882,A -85,B 0,C 180,E1 -8364.206,E2 -8364.206} C_VEL
LIN {X 0,Y 452.485,Z 398.499,A -85,B 0,C 180,E1 -8365.546,E2 -8365.546} C_VEL
LIN {X 0,Y 452.482,Z 400.365,A -85,B 0,C 180,E1 -8366.438,E2 -8366.438} C_VEL
LIN {X 0,Y 452.508,Z 401.766,A -85,B 0,C 180,E1 -8367.329,E2 -8367.329} C_VEL
LIN {X 0,Y 452.46,Z 403.372,A -85,B 0,C 180,E1 -8369.11,E2 -8369.11} C_VEL
LIN {X 0,Y 452.469,Z 403.59,A -85,B 0,C 180,E1 -8370,E2 -8370} C_VEL
LIN {X 0,Y 452.46,Z 403.372,A -85,B 0,C 180,E1 -8370.89,E2 -8370.89} C_VEL
LIN {X 0,Y 452.508,Z 401.767,A -85,B 0,C 180,E1 -8372.67,E2 -8372.67} C_VEL
LIN {X 0,Y 452.482,Z 400.366,A -85,B 0,C 180,E1 -8373.561,E2 -8373.561} C_VEL
LIN {X 0,Y 452.542,Z 397.424,A -85,B 0,C 180,E1 -8374.899,E2 -8374.899} C_VEL
LIN {X 0,Y 452.61,Z 392.903,A -85,B 0,C 180,E1 -8376.395,E2 -8376.395} C_VEL
LIN {X 0,Y 452.796,Z 387.318,A -85,B 0,C 180,E1 -8377.805,E2 -8377.805} C_VEL
LIN {X 0,Y 453.056,Z 380.628,A -85,B 0,C 180,E1 -8379.148,E2 -8379.148} C_VEL
LIN {X 0,Y 453.449,Z 372.331,A -85,B 0,C 180,E1 -8380.492,E2 -8380.492} C_VEL
LIN {X 0,Y 453.977,Z 363.833,A -85,B 0,C 180,E1 -8381.61,E2 -8381.61} C_VEL
LIN {X 0,Y 454.5,Z 354.212,A -85,B 0,C 180,E1 -8382.644,E2 -8382.644} C_VEL
LIN {X 0,Y 455.075,Z 342.945,A -85,B 0,C 180,E1 -8383.621,E2 -8383.621} C_VEL
LIN {X 0,Y 455.623,Z 331.56,A -85,B 0,C 180,E1 -8384.402,E2 -8384.402} C_VEL
LIN {X 0,Y 456.139,Z 319.884,A -85,B 0,C 180,E1 -8385.012,E2 -8385.012} C_VEL
LIN {X 0,Y 456.613,Z 307.347,A -85,B 0,C 180,E1 -8385.482,E2 -8385.482} C_VEL
LIN {X 0,Y 456.933,Z 294.651,A -85,B 0,C 180,E1 -8385.785,E2 -8385.785} C_VEL
LIN {X 0,Y 457.528,Z 211.296,A -85,B 0,C 180,E1 -8387.104,E2 -8387.104} C_VEL
LIN {X 0,Y 454.361,Z 190.674,A -85,B 0,C 180,E1 -8387.559,E2 -8387.559} C_VEL
LIN {X 0,Y 455.13,Z 172.444,A -85,B 0,C 180,E1 -8390.802,E2 -8390.802} C_VEL
LIN {X 0,Y 455.94,Z 156.742,A -85,B 0,C 180,E1 -8393.626,E2 -8393.626} C_VEL
LIN {X 0,Y 455.712,Z 153.062,A -85,B 0,C 180,E1 -8394.314,E2 -8394.314} C_VEL
LIN {X 0,Y 453.497,Z 141.997,A -85,B 0,C 180,E1 -8396.523,E2 -8396.523} C_VEL
LIN {X 0,Y 453.466,Z 142.003,A -85,B 0,C 180,E1 -8399.783,E2 -8399.783} C_VEL
LIN {X 0,Y 453.477,Z 141.997,A -85,B 0,C 180,E1 -8403.186,E2 -8403.186} C_VEL
LIN {X 0,Y 453.446,Z 141.998,A -85,B 0,C 180,E1 -8406.297,E2 -8406.297} C_VEL
LIN {X 0,Y 453.445,Z 142.005,A -85,B 0,C 180,E1 -8409.453,E2 -8409.453} C_VEL
LIN {X 0,Y 453.443,Z 141.999,A -85,B 0,C 180,E1 -8411.93,E2 -8411.93} C_VEL
LIN {X 0,Y 453.475,Z 141.998,A -85,B 0,C 180,E1 -8415.471,E2 -8415.471} C_VEL
LIN {X 0,Y 453.438,Z 141.998,A -85,B 0,C 180,E1 -8418.204,E2 -8418.204} C_VEL
LIN {X 0,Y 453.458,Z 142,A -85,B 0,C 180,E1 -8420.797,E2 -8420.797} C_VEL
LIN {X 0,Y 453.443,Z 141.998,A -85,B 0,C 180,E1 -8423.916,E2 -8423.916} C_VEL
LIN {X 0,Y 453.465,Z 141.999,A -85,B 0,C 180,E1 -8427.15,E2 -8427.15} C_VEL
LIN {X 0,Y 453.452,Z 141.998,A -85,B 0,C 180,E1 -8430.267,E2 -8430.267} C_VEL
LIN {X 0,Y 453.433,Z 142.001,A -85,B 0,C 180,E1 -8433.289,E2 -8433.289} C_VEL
LIN {X 0,Y 453.482,Z 141.996,A -85,B 0,C 180,E1 -8436.238,E2 -8436.238} C_VEL
LIN {X 0,Y 453.464,Z 141.997,A -85,B 0,C 180,E1 -8439.117,E2 -8439.117} C_VEL
LIN {X 0,Y 453.472,Z 141.996,A -85,B 0,C 180,E1 -8441.943,E2 -8441.943} C_VEL
LIN {X 0,Y 453.508,Z 141.993,A -85,B 0,C 180,E1 -8444.725,E2 -8444.725} C_VEL
LIN {X 0,Y 453.534,Z 141.993,A -85,B 0,C 180,E1 -8448.378,E2 -8448.378} C_VEL
LIN {X 0,Y 453.547,Z 141.985,A -85,B 0,C 180,E1 -8451.086,E2 -8451.086} C_VEL
LIN {X 0,Y 453.623,Z 141.979,A -85,B 0,C 180,E1 -8453.774,E2 -8453.774} C_VEL
LIN {X 0,Y 453.691,Z 141.968,A -85,B 0,C 180,E1 -8457.336,E2 -8457.336} C_VEL
LIN {X 0,Y 453.756,Z 141.966,A -85,B 0,C 180,E1 -8460,E2 -8460} C_VEL
LIN {X 0,Y 453.692,Z 141.967,A -85,B 0,C 180,E1 -8462.664,E2 -8462.664} C_VEL
LIN {X 0,Y 453.627,Z 141.977,A -85,B 0,C 180,E1 -8466.226,E2 -8466.226} C_VEL
LIN {X 0,Y 453.572,Z 141.982,A -85,B 0,C 180,E1 -8468.914,E2 -8468.914} C_VEL
LIN {X 0,Y 453.555,Z 141.984,A -85,B 0,C 180,E1 -8472.529,E2 -8472.529} C_VEL
LIN {X 0,Y 453.49,Z 141.993,A -85,B 0,C 180,E1 -8476.198,E2 -8476.198} C_VEL
LIN {X 0,Y 453.508,Z 141.993,A -85,B 0,C 180,E1 -8479.04,E2 -8479.04} C_VEL
LIN {X 0,Y 453.466,Z 141.997,A -85,B 0,C 180,E1 -8481.837,E2 -8481.837} C_VEL
LIN {X 0,Y 453.46,Z 141.997,A -85,B 0,C 180,E1 -8484.738,E2 -8484.738} C_VEL
LIN {X 0,Y 453.466,Z 141.995,A -85,B 0,C 180,E1 -8487.946,E2 -8487.946} C_VEL
LIN {X 0,Y 453.466,Z 141.998,A -85,B 0,C 180,E1 -8490.76,E2 -8490.76} C_VEL
LIN {X 0,Y 453.459,Z 141.996,A -85,B 0,C 180,E1 -8493.914,E2 -8493.914} C_VEL
LIN {X 0,Y 453.445,Z 142.002,A -85,B 0,C 180,E1 -8497.191,E2 -8497.191} C_VEL
LIN {X 0,Y 453.464,Z 142,A -85,B 0,C 180,E1 -8500.612,E2 -8500.612} C_VEL
LIN {X 0,Y 453.453,Z 141.998,A -85,B 0,C 180,E1 -8504.223,E2 -8504.223} C_VEL
LIN {X 0,Y 453.444,Z 142.001,A -85,B 0,C 180,E1 -8507.004,E2 -8507.004} C_VEL
LIN {X 0,Y 453.489,Z 141.992,A -85,B 0,C 180,E1 -8509.41,E2 -8509.41} C_VEL
LIN {X 0,Y 453.446,Z 142.001,A -85,B 0,C 180,E1 -8512.811,E2 -8512.811} C_VEL
LIN {X 0,Y 453.474,Z 141.998,A -85,B 0,C 180,E1 -8516.088,E2 -8516.088} C_VEL
LIN {X 0,Y 453.472,Z 141.994,A -85,B 0,C 180,E1 -8519.241,E2 -8519.241} C_VEL
LIN {X 0,Y 453.495,Z 141.998,A -85,B 0,C 180,E1 -8522.296,E2 -8522.296} C_VEL
LIN {X 0,Y 453.493,Z 141.992,A -85,B 0,C 180,E1 -8525.265,E2 -8525.265} C_VEL
LIN {X 0,Y 453.5,Z 142.026,A -85,B 0,C 180,E1 -8528.727,E2 -8528.727} C_VEL
LIN {X 0,Y 454.911,Z 149.788,A -85,B 0,C 180,E1 -8530.459,E2 -8530.459} C_VEL
LIN {X 0,Y 454.653,Z 159.837,A -85,B 0,C 180,E1 -8532.511,E2 -8532.511} C_VEL
LIN {X 0,Y 457.879,Z 176.098,A -85,B 0,C 180,E1 -8532.903,E2 -8532.903} C_VEL
LIN {X 0,Y 457.574,Z 216.54,A -85,B 0,C 180,E1 -8533.541,E2 -8533.541} C_VEL
LIN {X 0,Y 456.922,Z 222.379,A -85,B 0,C 180,E1 -8533.61,E2 -8533.61} C_VEL
LIN {X 0,Y 451.241,Z 241.364,A -85,B 0,C 180,E1 -8533.703,E2 -8533.703} C_VEL
LIN {X 0,Y 450.539,Z 247.206,A -85,B 0,C 180,E1 -8533.772,E2 -8533.772} C_VEL
LIN {X 0,Y 450.182,Z 268.785,A -85,B 0,C 180,E1 -8534.146,E2 -8534.146} C_VEL
LIN {X 0,Y 449.863,Z 282.259,A -85,B 0,C 180,E1 -8534.57,E2 -8534.57} C_VEL
LIN {X 0,Y 449.385,Z 294.9,A -85,B 0,C 180,E1 -8535.162,E2 -8535.162} C_VEL
LIN {X 0,Y 448.863,Z 307.321,A -85,B 0,C 180,E1 -8535.956,E2 -8535.956} C_VEL
LIN {X 0,Y 448.438,Z 318.369,A -85,B 0,C 180,E1 -8536.866,E2 -8536.866} C_VEL
LIN {X 0,Y 447.793,Z 327.322,A -85,B 0,C 180,E1 -8537.768,E2 -8537.768} C_VEL
LIN {X 0,Y 447.29,Z 336.497,A -85,B 0,C 180,E1 -8538.903,E2 -8538.903} C_VEL
LIN {X 0,Y 446.714,Z 345.404,A -85,B 0,C 180,E1 -8540.264,E2 -8540.264} C_VEL
LIN {X 0,Y 446.246,Z 352.574,A -85,B 0,C 180,E1 -8541.624,E2 -8541.624} C_VEL
LIN {X 0,Y 445.929,Z 358.958,A -85,B 0,C 180,E1 -8543.171,E2 -8543.171} C_VEL
LIN {X 0,Y 445.675,Z 363.419,A -85,B 0,C 180,E1 -8544.571,E2 -8544.571} C_VEL
LIN {X 0,Y 445.572,Z 365.702,A -85,B 0,C 180,E1 -8545.477,E2 -8545.477} C_VEL
LIN {X 0,Y 445.618,Z 367.556,A -85,B 0,C 180,E1 -8546.384,E2 -8546.384} C_VEL
LIN {X 0,Y 445.496,Z 368.959,A -85,B 0,C 180,E1 -8547.288,E2 -8547.288} C_VEL
LIN {X 0,Y 445.373,Z 370.57,A -85,B 0,C 180,E1 -8549.096,E2 -8549.096} C_VEL
LIN {X 0,Y 445.378,Z 370.804,A -85,B 0,C 180,E1 -8550,E2 -8550} C_VEL
LIN {X 0,Y 445.373,Z 370.618,A -85,B 0,C 180,E1 -8550.905,E2 -8550.905} C_VEL
LIN {X 0,Y 445.496,Z 369.07,A -85,B 0,C 180,E1 -8552.713,E2 -8552.713} C_VEL
LIN {X 0,Y 445.6,Z 367.716,A -85,B 0,C 180,E1 -8553.617,E2 -8553.617} C_VEL
LIN {X 0,Y 445.59,Z 364.862,A -85,B 0,C 180,E1 -8554.977,E2 -8554.977} C_VEL
LIN {X 0,Y 445.899,Z 360.98,A -85,B 0,C 180,E1 -8556.335,E2 -8556.335} C_VEL
LIN {X 0,Y 446.031,Z 355.981,A -85,B 0,C 180,E1 -8557.697,E2 -8557.697} C_VEL
LIN {X 0,Y 446.442,Z 349.681,A -85,B 0,C 180,E1 -8559.058,E2 -8559.058} C_VEL
LIN {X 0,Y 446.902,Z 341.794,A -85,B 0,C 180,E1 -8560.42,E2 -8560.42} C_VEL
LIN {X 0,Y 447.521,Z 331.978,A -85,B 0,C 180,E1 -8561.78,E2 -8561.78} C_VEL
LIN {X 0,Y 448.222,Z 321.714,A -85,B 0,C 180,E1 -8562.907,E2 -8562.907} C_VEL
LIN {X 0,Y 448.729,Z 310.234,A -85,B 0,C 180,E1 -8563.92,E2 -8563.92} C_VEL
LIN {X 0,Y 449.277,Z 298.483,A -85,B 0,C 180,E1 -8564.726,E2 -8564.726} C_VEL
LIN {X 0,Y 449.746,Z 286.444,A -85,B 0,C 180,E1 -8565.348,E2 -8565.348} C_VEL
LIN {X 0,Y 450.153,Z 273.324,A -85,B 0,C 180,E1 -8565.827,E2 -8565.827} C_VEL
LIN {X 0,Y 450.433,Z 260.662,A -85,B 0,C 180,E1 -8566.108,E2 -8566.108} C_VEL
LIN {X 0,Y 451.011,Z 176.757,A -85,B 0,C 180,E1 -8567.455,E2 -8567.455} C_VEL
LIN {X 0,Y 447.686,Z 159.953,A -85,B 0,C 180,E1 -8567.873,E2 -8567.873} C_VEL
LIN {X 0,Y 447.884,Z 150.344,A -85,B 0,C 180,E1 -8569.884,E2 -8569.884} C_VEL
LIN {X 0,Y 446.446,Z 142.876,A -85,B 0,C 180,E1 -8571.588,E2 -8571.588} C_VEL
LIN {X 0,Y 446.464,Z 142.873,A -85,B 0,C 180,E1 -8574.16,E2 -8574.16} C_VEL
LIN {X 0,Y 446.447,Z 142.87,A -85,B 0,C 180,E1 -8577.163,E2 -8577.163} C_VEL
LIN {X 0,Y 446.427,Z 142.874,A -85,B 0,C 180,E1 -8580.25,E2 -8580.25} C_VEL
LIN {X 0,Y 446.447,Z 142.874,A -85,B 0,C 180,E1 -8583.453,E2 -8583.453} C_VEL
LIN {X 0,Y 446.401,Z 142.875,A -85,B 0,C 180,E1 -8586.745,E2 -8586.745} C_VEL
LIN {X 0,Y 446.402,Z 142.883,A -85,B 0,C 180,E1 -8589.516,E2 -8589.516} C_VEL
LIN {X 0,Y 446.416,Z 142.873,A -85,B 0,C 180,E1 -8592.606,E2 -8592.606} C_VEL
LIN {X 0,Y 446.45,Z 142.873,A -85,B 0,C 180,E1 -8595.104,E2 -8595.104} C_VEL
LIN {X 0,Y 446.41,Z 142.875,A -85,B 0,C 180,E1 -8598.607,E2 -8598.607} C_VEL
LIN {X 0,Y 446.409,Z 142.875,A -85,B 0,C 180,E1 -8601.921,E2 -8601.921} C_VEL
LIN {X 0,Y 446.42,Z 142.875,A -85,B 0,C 180,E1 -8605.476,E2 -8605.476} C_VEL
LIN {X 0,Y 446.408,Z 142.878,A -85,B 0,C 180,E1 -8608.699,E2 -8608.699} C_VEL
LIN {X 0,Y 446.445,Z 142.87,A -85,B 0,C 180,E1 -8611.83,E2 -8611.83} C_VEL
LIN {X 0,Y 446.436,Z 142.878,A -85,B 0,C 180,E1 -8614.846,E2 -8614.846} C_VEL
LIN {X 0,Y 446.446,Z 142.872,A -85,B 0,C 180,E1 -8618.245,E2 -8618.245} C_VEL
LIN {X 0,Y 446.436,Z 142.871,A -85,B 0,C 180,E1 -8621.648,E2 -8621.648} C_VEL
LIN {X 0,Y 446.456,Z 142.876,A -85,B 0,C 180,E1 -8624.478,E2 -8624.478} C_VEL
LIN {X 0,Y 446.514,Z 142.861,A -85,B 0,C 180,E1 -8627.384,E2 -8627.384} C_VEL
LIN {X 0,Y 446.522,Z 142.861,A -85,B 0,C 180,E1 -8630.944,E2 -8630.944} C_VEL
LIN {X 0,Y 446.6,Z 142.852,A -85,B 0,C 180,E1 -8633.676,E2 -8633.676} C_VEL
LIN {X 0,Y 446.648,Z 142.844,A -85,B 0,C 180,E1 -8637.294,E2 -8637.294} C_VEL
LIN {X 0,Y 446.714,Z 142.843,A -85,B 0,C 180,E1 -8640,E2 -8640} C_VEL
LIN {X 0,Y 446.646,Z 142.845,A -85,B 0,C 180,E1 -8642.706,E2 -8642.706} C_VEL
LIN {X 0,Y 446.599,Z 142.853,A -85,B 0,C 180,E1 -8646.324,E2 -8646.324} C_VEL
LIN {X 0,Y 446.502,Z 142.863,A -85,B 0,C 180,E1 -8649.056,E2 -8649.056} C_VEL
LIN {X 0,Y 446.489,Z 142.864,A -85,B 0,C 180,E1 -8652.731,E2 -8652.731} C_VEL
LIN {X 0,Y 446.451,Z 142.87,A -85,B 0,C 180,E1 -8656.209,E2 -8656.209} C_VEL
LIN {X 0,Y 446.428,Z 142.877,A -85,B 0,C 180,E1 -8659.305,E2 -8659.305} C_VEL
LIN {X 0,Y 446.403,Z 142.875,A -85,B 0,C 180,E1 -8662.2,E2 -8662.2} C_VEL
LIN {X 0,Y 446.417,Z 142.878,A -85,B 0,C 180,E1 -8665.155,E2 -8665.155} C_VEL
LIN {X 0,Y 446.413,Z 142.874,A -85,B 0,C 180,E1 -8668.184,E2 -8668.184} C_VEL
LIN {X 0,Y 446.388,Z 142.883,A -85,B 0,C 180,E1 -8671.303,E2 -8671.303} C_VEL
LIN {X 0,Y 446.419,Z 142.874,A -85,B 0,C 180,E1 -8674.524,E2 -8674.524} C_VEL
LIN {X 0,Y 446.408,Z 142.874,A -85,B 0,C 180,E1 -8678.078,E2 -8678.078} C_VEL
LIN {X 0,Y 446.399,Z 142.877,A -85,B 0,C 180,E1 -8681.395,E2 -8681.395} C_VEL
LIN {X 0,Y 446.448,Z 142.873,A -85,B 0,C 180,E1 -8685.104,E2 -8685.104} C_VEL
LIN {X 0,Y 446.4,Z 142.882,A -85,B 0,C 180,E1 -8688.606,E2 -8688.606} C_VEL
LIN {X 0,Y 446.41,Z 142.875,A -85,B 0,C 180,E1 -8691.922,E2 -8691.922} C_VEL
LIN {X 0,Y 446.422,Z 142.872,A -85,B 0,C 180,E1 -8695.476,E2 -8695.476} C_VEL
LIN {X 0,Y 446.415,Z 142.879,A -85,B 0,C 180,E1 -8698.7,E2 -8698.7} C_VEL
LIN {X 0,Y 446.448,Z 142.875,A -85,B 0,C 180,E1 -8701.831,E2 -8701.831} C_VEL
LIN {X 0,Y 446.482,Z 143.026,A -85,B 0,C 180,E1 -8703.299,E2 -8703.299} C_VEL
LIN {X 0,Y 448.858,Z 154.876,A -85,B 0,C 180,E1 -8705.673,E2 -8705.673} C_VEL
LIN {X 0,Y 448.912,Z 160.439,A -85,B 0,C 180,E1 -8706.715,E2 -8706.715} C_VEL
LIN {X 0,Y 447.866,Z 180.192,A -85,B 0,C 180,E1 -8710.311,E2 -8710.311} C_VEL
LIN {X 0,Y 447.351,Z 190.281,A -85,B 0,C 180,E1 -8712.129,E2 -8712.129} C_VEL
LIN {X 0,Y 450.788,Z 212.968,A -85,B 0,C 180,E1 -8712.66,E2 -8712.66} C_VEL
LIN {X 0,Y 450.032,Z 298.874,A -85,B 0,C 180,E1 -8714.052,E2 -8714.052} C_VEL
LIN {X 0,Y 449.617,Z 312.137,A -85,B 0,C 180,E1 -8714.444,E2 -8714.444} C_VEL
LIN {X 0,Y 449.025,Z 325.419,A -85,B 0,C 180,E1 -8715.033,E2 -8715.033} C_VEL
LIN {X 0,Y 448.452,Z 336.572,A -85,B 0,C 180,E1 -8715.71,E2 -8715.71} C_VEL
LIN {X 0,Y 447.876,Z 347.211,A -85,B 0,C 180,E1 -8716.531,E2 -8716.531} C_VEL
LIN {X 0,Y 447.288,Z 358.634,A -85,B 0,C 180,E1 -8717.638,E2 -8717.638} C_VEL
LIN {X 0,Y 446.785,Z 367.183,A -85,B 0,C 180,E1 -8718.66,E2 -8718.66} C_VEL
LIN {X 0,Y 446.304,Z 375.072,A -85,B 0,C 180,E1 -8719.796,E2 -8719.796} C_VEL
LIN {X 0,Y 445.914,Z 382.782,A -85,B 0,C 180,E1 -8721.16,E2 -8721.16} C_VEL
LIN {X 0,Y 445.602,Z 389.891,A -85,B 0,C 180,E1 -8722.751,E2 -8722.751} C_VEL
LIN {X 0,Y 445.445,Z 394.218,A -85,B 0,C 180,E1 -8723.985,E2 -8723.985} C_VEL
LIN {X 0,Y 445.411,Z 398.241,A -85,B 0,C 180,E1 -8725.475,E2 -8725.475} C_VEL
LIN {X 0,Y 445.38,Z 400.106,A -85,B 0,C 180,E1 -8726.381,E2 -8726.381} C_VEL
LIN {X 0,Y 445.433,Z 401.508,A -85,B 0,C 180,E1 -8727.287,E2 -8727.287} C_VEL
LIN {X 0,Y 445.368,Z 403.114,A -85,B 0,C 180,E1 -8729.095,E2 -8729.095} C_VEL
LIN {X 0,Y 445.375,Z 403.331,A -85,B 0,C 180,E1 -8730,E2 -8730} C_VEL
LIN {X 0,Y 445.368,Z 403.113,A -85,B 0,C 180,E1 -8730.904,E2 -8730.904} C_VEL
LIN {X 0,Y 445.433,Z 401.508,A -85,B 0,C 180,E1 -8732.713,E2 -8732.713} C_VEL
LIN {X 0,Y 445.38,Z 400.106,A -85,B 0,C 180,E1 -8733.618,E2 -8733.618} C_VEL
LIN {X 0,Y 445.471,Z 397.165,A -85,B 0,C 180,E1 -8734.977,E2 -8734.977} C_VEL
LIN {X 0,Y 445.555,Z 391.745,A -85,B 0,C 180,E1 -8736.748,E2 -8736.748} C_VEL
LIN {X 0,Y 445.754,Z 386.041,A -85,B 0,C 180,E1 -8738.157,E2 -8738.157} C_VEL
LIN {X 0,Y 446.06,Z 379.126,A -85,B 0,C 180,E1 -8739.522,E2 -8739.522} C_VEL
LIN {X 0,Y 446.524,Z 370.479,A -85,B 0,C 180,E1 -8740.886,E2 -8740.886} C_VEL
LIN {X 0,Y 447.114,Z 361.617,A -85,B 0,C 180,E1 -8742.02,E2 -8742.02} C_VEL
LIN {X 0,Y 447.695,Z 351.161,A -85,B 0,C 180,E1 -8743.112,E2 -8743.112} C_VEL
LIN {X 0,Y 448.273,Z 339.706,A -85,B 0,C 180,E1 -8744.063,E2 -8744.063} C_VEL
LIN {X 0,Y 448.936,Z 327.377,A -85,B 0,C 180,E1 -8744.853,E2 -8744.853} C_VEL
LIN {X 0,Y 449.48,Z 315.711,A -85,B 0,C 180,E1 -8745.414,E2 -8745.414} C_VEL
LIN {X 0,Y 449.94,Z 303.307,A -85,B 0,C 180,E1 -8745.834,E2 -8745.834} C_VEL
LIN {X 0,Y 450.206,Z 287.49,A -85,B 0,C 180,E1 -8746.144,E2 -8746.144} C_VEL
LIN {X 0,Y 450.682,Z 211.826,A -85,B 0,C 180,E1 -8747.358,E2 -8747.358} C_VEL
LIN {X 0,Y 447.398,Z 190.308,A -85,B 0,C 180,E1 -8747.86,E2 -8747.86} C_VEL
LIN {X 0,Y 448.235,Z 172.181,A -85,B 0,C 180,E1 -8751.138,E2 -8751.138} C_VEL
LIN {X 0,Y 449.044,Z 156.48,A -85,B 0,C 180,E1 -8754.011,E2 -8754.011} C_VEL
LIN {X 0,Y 446.861,Z 144.963,A -85,B 0,C 180,E1 -8756.302,E2 -8756.302} C_VEL
LIN {X 0,Y 446.459,Z 142.874,A -85,B 0,C 180,E1 -8756.731,E2 -8756.731} C_VEL
LIN {X 0,Y 446.426,Z 142.878,A -85,B 0,C 180,E1 -8760.019,E2 -8760.019} C_VEL
LIN {X 0,Y 446.42,Z 142.879,A -85,B 0,C 180,E1 -8763.448,E2 -8763.448} C_VEL
LIN {X 0,Y 446.396,Z 142.876,A -85,B 0,C 180,E1 -8766.745,E2 -8766.745} C_VEL
LIN {X 0,Y 446.397,Z 142.881,A -85,B 0,C 180,E1 -8769.516,E2 -8769.516} C_VEL
LIN {X 0,Y 446.382,Z 142.878,A -85,B 0,C 180,E1 -8772.609,E2 -8772.609} C_VEL
LIN {X 0,Y 446.444,Z 142.876,A -85,B 0,C 180,E1 -8775.103,E2 -8775.103} C_VEL
LIN {X 0,Y 446.395,Z 142.878,A -85,B 0,C 180,E1 -8778.605,E2 -8778.605} C_VEL
LIN {X 0,Y 446.403,Z 142.875,A -85,B 0,C 180,E1 -8781.921,E2 -8781.921} C_VEL
LIN {X 0,Y 446.414,Z 142.875,A -85,B 0,C 180,E1 -8785.476,E2 -8785.476} C_VEL
LIN {X 0,Y 446.399,Z 142.881,A -85,B 0,C 180,E1 -8788.698,E2 -8788.698} C_VEL
LIN {X 0,Y 446.415,Z 142.873,A -85,B 0,C 180,E1 -8791.836,E2 -8791.836} C_VEL
LIN {X 0,Y 446.412,Z 142.879,A -85,B 0,C 180,E1 -8794.845,E2 -8794.845} C_VEL
LIN {X 0,Y 446.437,Z 142.874,A -85,B 0,C 180,E1 -8798.245,E2 -8798.245} C_VEL
LIN {X 0,Y 446.428,Z 142.872,A -85,B 0,C 180,E1 -8801.648,E2 -8801.648} C_VEL
LIN {X 0,Y 446.447,Z 142.876,A -85,B 0,C 180,E1 -8804.478,E2 -8804.478} C_VEL
LIN {X 0,Y 446.506,Z 142.862,A -85,B 0,C 180,E1 -8807.384,E2 -8807.384} C_VEL
LIN {X 0,Y 446.498,Z 142.864,A -85,B 0,C 180,E1 -8810.944,E2 -8810.944} C_VEL
LIN {X 0,Y 446.593,Z 142.853,A -85,B 0,C 180,E1 -8813.676,E2 -8813.676} C_VEL
LIN {X 0,Y 446.64,Z 142.846,A -85,B 0,C 180,E1 -8817.294,E2 -8817.294} C_VEL
LIN {X 0,Y 446.707,Z 142.844,A -85,B 0,C 180,E1 -8820,E2 -8820} C_VEL
LIN {X 0,Y 446.642,Z 142.845,A -85,B 0,C 180,E1 -8822.706,E2 -8822.706} C_VEL
LIN {X 0,Y 446.597,Z 142.852,A -85,B 0,C 180,E1 -8826.324,E2 -8826.324} C_VEL
LIN {X 0,Y 446.52,Z 142.861,A -85,B 0,C 180,E1 -8829.056,E2 -8829.056} C_VEL
LIN {X 0,Y 446.512,Z 142.861,A -85,B 0,C 180,E1 -8832.73,E2 -8832.73} C_VEL
LIN {X 0,Y 446.444,Z 142.87,A -85,B 0,C 180,E1 -8836.209,E2 -8836.209} C_VEL
LIN {X 0,Y 446.459,Z 142.874,A -85,B 0,C 180,E1 -8839.304,E2 -8839.304} C_VEL
LIN {X 0,Y 446.407,Z 142.874,A -85,B 0,C 180,E1 -8842.2,E2 -8842.2} C_VEL
LIN {X 0,Y 446.412,Z 142.88,A -85,B 0,C 180,E1 -8845.155,E2 -8845.155} C_VEL
LIN {X 0,Y 446.43,Z 142.872,A -85,B 0,C 180,E1 -8848.183,E2 -8848.183} C_VEL
LIN {X 0,Y 446.406,Z 142.879,A -85,B 0,C 180,E1 -8851.301,E2 -8851.301} C_VEL
LIN {X 0,Y 446.415,Z 142.875,A -85,B 0,C 180,E1 -8854.524,E2 -8854.524} C_VEL
LIN {X 0,Y 446.405,Z 142.875,A -85,B 0,C 180,E1 -8858.079,E2 -8858.079} C_VEL
LIN {X 0,Y 446.399,Z 142.877,A -85,B 0,C 180,E1 -8861.395,E2 -8861.395} C_VEL
LIN {X 0,Y 446.445,Z 142.873,A -85,B 0,C 180,E1 -8865.105,E2 -8865.105} C_VEL
LIN {X 0,Y 446.414,Z 142.881,A -85,B 0,C 180,E1 -8868.609,E2 -8868.609} C_VEL
LIN {X 0,Y 446.407,Z 142.876,A -85,B 0,C 180,E1 -8871.923,E2 -8871.923} C_VEL
LIN {X 0,Y 446.426,Z 142.872,A -85,B 0,C 180,E1 -8875.478,E2 -8875.478} C_VEL
LIN {X 0,Y 446.413,Z 142.877,A -85,B 0,C 180,E1 -8878.7,E2 -8878.7} C_VEL
LIN {X 0,Y 446.446,Z 142.872,A -85,B 0,C 180,E1 -8881.831,E2 -8881.831} C_VEL
LIN {X 0,Y 446.437,Z 142.871,A -85,B 0,C 180,E1 -8884.847,E2 -8884.847} C_VEL
LIN {X 0,Y 446.449,Z 142.876,A -85,B 0,C 180,E1 -8888.246,E2 -8888.246} C_VEL
LIN {X 0,Y 446.47,Z 142.981,A -85,B 0,C 180,E1 -8888.544,E2 -8888.544} C_VEL
LIN {X 0,Y 447.919,Z 150.708,A -85,B 0,C 180,E1 -8890.292,E2 -8890.292} C_VEL
LIN {X 0,Y 447.699,Z 159.917,A -85,B 0,C 180,E1 -8892.216,E2 -8892.216} C_VEL
LIN {X 0,Y 451.114,Z 177.367,A -85,B 0,C 180,E1 -8892.654,E2 -8892.654} C_VEL
LIN {X 0,Y 450.539,Z 247.206,A -85,B 0,C 180,E1 -8893.772,E2 -8893.772} C_VEL
LIN {X 0,Y 449.828,Z 253.046,A -85,B 0,C 180,E1 -8893.837,E2 -8893.837} C_VEL
LIN {X 0,Y 444.443,Z 270.038,A -85,B 0,C 180,E1 -8893.962,E2 -8893.962} C_VEL
LIN {X 0,Y 443.329,Z 275.752,A -85,B 0,C 180,E1 -8894.088,E2 -8894.088} C_VEL
LIN {X 0,Y 443.211,Z 277.666,A -85,B 0,C 180,E1 -8894.147,E2 -8894.147} C_VEL
LIN {X 0,Y 442.796,Z 289.674,A -85,B 0,C 180,E1 -8894.642,E2 -8894.642} C_VEL
LIN {X 0,Y 442.314,Z 300.91,A -85,B 0,C 180,E1 -8895.273,E2 -8895.273} C_VEL
LIN {X 0,Y 441.755,Z 311.581,A -85,B 0,C 180,E1 -8896.041,E2 -8896.041} C_VEL
LIN {X 0,Y 441.28,Z 322.2,A -85,B 0,C 180,E1 -8897.004,E2 -8897.004} C_VEL
LIN {X 0,Y 440.602,Z 331.485,A -85,B 0,C 180,E1 -8898.033,E2 -8898.033} C_VEL
LIN {X 0,Y 440.087,Z 339.976,A -85,B 0,C 180,E1 -8899.185,E2 -8899.185} C_VEL
LIN {X 0,Y 439.536,Z 348.224,A -85,B 0,C 180,E1 -8900.568,E2 -8900.568} C_VEL
LIN {X 0,Y 439.14,Z 353.867,A -85,B 0,C 180,E1 -8901.719,E2 -8901.719} C_VEL
LIN {X 0,Y 438.875,Z 359.511,A -85,B 0,C 180,E1 -8903.146,E2 -8903.146} C_VEL
LIN {X 0,Y 438.631,Z 363.678,A -85,B 0,C 180,E1 -8904.484,E2 -8904.484} C_VEL
LIN {X 0,Y 438.489,Z 365.962,A -85,B 0,C 180,E1 -8905.404,E2 -8905.404} C_VEL
LIN {X 0,Y 438.535,Z 367.816,A -85,B 0,C 180,E1 -8906.325,E2 -8906.325} C_VEL
LIN {X 0,Y 438.427,Z 369.218,A -85,B 0,C 180,E1 -8907.244,E2 -8907.244} C_VEL
LIN {X 0,Y 438.285,Z 370.829,A -85,B 0,C 180,E1 -8909.082,E2 -8909.082} C_VEL
LIN {X 0,Y 438.287,Z 371.063,A -85,B 0,C 180,E1 -8910,E2 -8910} C_VEL
LIN {X 0,Y 438.285,Z 370.877,A -85,B 0,C 180,E1 -8910.919,E2 -8910.919} C_VEL
LIN {X 0,Y 438.427,Z 369.327,A -85,B 0,C 180,E1 -8912.757,E2 -8912.757} C_VEL
LIN {X 0,Y 438.518,Z 367.974,A -85,B 0,C 180,E1 -8913.676,E2 -8913.676} C_VEL
LIN {X 0,Y 438.527,Z 365.119,A -85,B 0,C 180,E1 -8915.057,E2 -8915.057} C_VEL
LIN {X 0,Y 438.813,Z 361.239,A -85,B 0,C 180,E1 -8916.437,E2 -8916.437} C_VEL
LIN {X 0,Y 439.004,Z 356.238,A -85,B 0,C 180,E1 -8917.821,E2 -8917.821} C_VEL
LIN {X 0,Y 439.441,Z 349.938,A -85,B 0,C 180,E1 -8919.203,E2 -8919.203} C_VEL
LIN {X 0,Y 439.912,Z 342.05,A -85,B 0,C 180,E1 -8920.587,E2 -8920.587} C_VEL
LIN {X 0,Y 440.592,Z 332.233,A -85,B 0,C 180,E1 -8921.968,E2 -8921.968} C_VEL
LIN {X 0,Y 441.31,Z 322.12,A -85,B 0,C 180,E1 -8923.098,E2 -8923.098} C_VEL
LIN {X 0,Y 441.795,Z 311.732,A -85,B 0,C 180,E1 -8924.04,E2 -8924.04} C_VEL
LIN {X 0,Y 442.369,Z 300.557,A -85,B 0,C 180,E1 -8924.844,E2 -8924.844} C_VEL
LIN {X 0,Y 442.833,Z 289.228,A -85,B 0,C 180,E1 -8925.476,E2 -8925.476} C_VEL
LIN {X 0,Y 443.261,Z 276.312,A -85,B 0,C 180,E1 -8925.991,E2 -8925.991} C_VEL
LIN {X 0,Y 443.583,Z 262.508,A -85,B 0,C 180,E1 -8926.334,E2 -8926.334} C_VEL
LIN {X 0,Y 444.3,Z 177.875,A -85,B 0,C 180,E1 -8927.712,E2 -8927.712} C_VEL
LIN {X 0,Y 440.779,Z 160.199,A -85,B 0,C 180,E1 -8928.163,E2 -8928.163} C_VEL
LIN {X 0,Y 440.98,Z 151.999,A -85,B 0,C 180,E1 -8929.898,E2 -8929.898} C_VEL
LIN {X 0,Y 439.4,Z 143.753,A -85,B 0,C 180,E1 -8931.817,E2 -8931.817} C_VEL
LIN {X 0,Y 439.41,Z 143.749,A -85,B 0,C 180,E1 -8934.573,E2 -8934.573} C_VEL
LIN {X 0,Y 439.388,Z 143.753,A -85,B 0,C 180,E1 -8937.636,E2 -8937.636} C_VEL
LIN {X 0,Y 439.362,Z 143.752,A -85,B 0,C 180,E1 -8940.788,E2 -8940.788} C_VEL
LIN {X 0,Y 439.389,Z 143.752,A -85,B 0,C 180,E1 -8944.044,E2 -8944.044} C_VEL
LIN {X 0,Y 439.347,Z 143.754,A -85,B 0,C 180,E1 -8946.886,E2 -8946.886} C_VEL
LIN {X 0,Y 439.349,Z 143.757,A -85,B 0,C 180,E1 -8949.84,E2 -8949.84} C_VEL
LIN {X 0,Y 439.37,Z 143.751,A -85,B 0,C 180,E1 -8952.625,E2 -8952.625} C_VEL
LIN {X 0,Y 439.398,Z 143.754,A -85,B 0,C 180,E1 -8955.27,E2 -8955.27} C_VEL
LIN {X 0,Y 439.37,Z 143.753,A -85,B 0,C 180,E1 -8958.746,E2 -8958.746} C_VEL
LIN {X 0,Y 439.366,Z 143.754,A -85,B 0,C 180,E1 -8961.609,E2 -8961.609} C_VEL
LIN {X 0,Y 439.394,Z 143.753,A -85,B 0,C 180,E1 -8964.843,E2 -8964.843} C_VEL
LIN {X 0,Y 439.364,Z 143.752,A -85,B 0,C 180,E1 -8968.139,E2 -8968.139} C_VEL
LIN {X 0,Y 439.399,Z 143.748,A -85,B 0,C 180,E1 -8971.606,E2 -8971.606} C_VEL
LIN {X 0,Y 439.374,Z 143.753,A -85,B 0,C 180,E1 -8974.413,E2 -8974.413} C_VEL
LIN {X 0,Y 439.361,Z 143.753,A -85,B 0,C 180,E1 -8977.424,E2 -8977.424} C_VEL
LIN {X 0,Y 439.439,Z 143.75,A -85,B 0,C 180,E1 -8980.663,E2 -8980.663} C_VEL
LIN {X 0,Y 439.416,Z 143.749,A -85,B 0,C 180,E1 -8984.223,E2 -8984.223} C_VEL
LIN {X 0,Y 439.482,Z 143.737,A -85,B 0,C 180,E1 -8987.285,E2 -8987.285} C_VEL
LIN {X 0,Y 439.486,Z 143.739,A -85,B 0,C 180,E1 -8990.798,E2 -8990.798} C_VEL
LIN {X 0,Y 439.554,Z 143.729,A -85,B 0,C 180,E1 -8993.574,E2 -8993.574} C_VEL
LIN {X 0,Y 439.401,Z 143.747,A -85,B 0,C 180,E1 -8995.413,E2 -8995.413} C_VEL
LIN {X 0,Y 439.622,Z 143.727,A -85,B 0,C 180,E1 -8998.168,E2 -8998.168} C_VEL
LIN {X 0,Y 439.665,Z 143.721,A -85,B 0,C 180,E1 -9000,E2 -9000} C_VEL
LIN {X 0,Y 439.598,Z 143.723,A -85,B 0,C 180,E1 -9002.749,E2 -9002.749} C_VEL
LIN {X 0,Y 439.553,Z 143.73,A -85,B 0,C 180,E1 -9006.426,E2 -9006.426} C_VEL
LIN {X 0,Y 439.468,Z 143.74,A -85,B 0,C 180,E1 -9009.202,E2 -9009.202} C_VEL
LIN {X 0,Y 439.448,Z 143.742,A -85,B 0,C 180,E1 -9012.938,E2 -9012.938} C_VEL
LIN {X 0,Y 439.393,Z 143.749,A -85,B 0,C 180,E1 -9016.325,E2 -9016.325} C_VEL
LIN {X 0,Y 439.374,Z 143.757,A -85,B 0,C 180,E1 -9019.628,E2 -9019.628} C_VEL
LIN {X 0,Y 439.349,Z 143.754,A -85,B 0,C 180,E1 -9022.576,E2 -9022.576} C_VEL
LIN {X 0,Y 439.363,Z 143.756,A -85,B 0,C 180,E1 -9025.588,E2 -9025.588} C_VEL
LIN {X 0,Y 439.374,Z 143.752,A -85,B 0,C 180,E1 -9028.677,E2 -9028.677} C_VEL
LIN {X 0,Y 439.349,Z 143.754,A -85,B 0,C 180,E1 -9032.026,E2 -9032.026} C_VEL
LIN {X 0,Y 439.388,Z 143.753,A -85,B 0,C 180,E1 -9035.339,E2 -9035.339} C_VEL
LIN {X 0,Y 439.366,Z 143.755,A -85,B 0,C 180,E1 -9038.597,E2 -9038.597} C_VEL
LIN {X 0,Y 439.362,Z 143.755,A -85,B 0,C 180,E1 -9041.253,E2 -9041.253} C_VEL
LIN {X 0,Y 439.396,Z 143.755,A -85,B 0,C 180,E1 -9044.73,E2 -9044.73} C_VEL
LIN {X 0,Y 439.348,Z 143.754,A -85,B 0,C 180,E1 -9047.79,E2 -9047.79} C_VEL
LIN {X 0,Y 439.362,Z 143.752,A -85,B 0,C 180,E1 -9051.403,E2 -9051.403} C_VEL
LIN {X 0,Y 439.395,Z 143.751,A -85,B 0,C 180,E1 -9054.844,E2 -9054.844} C_VEL
LIN {X 0,Y 439.37,Z 143.755,A -85,B 0,C 180,E1 -9058.139,E2 -9058.139} C_VEL
LIN {X 0,Y 439.402,Z 143.751,A -85,B 0,C 180,E1 -9061.606,E2 -9061.606} C_VEL
LIN {X 0,Y 439.426,Z 143.825,A -85,B 0,C 180,E1 -9063.043,E2 -9063.043} C_VEL
LIN {X 0,Y 441.905,Z 156.239,A -85,B 0,C 180,E1 -9065.575,E2 -9065.575} C_VEL
LIN {X 0,Y 441.983,Z 161.49,A -85,B 0,C 180,E1 -9066.576,E2 -9066.576} C_VEL
LIN {X 0,Y 440.886,Z 180.735,A -85,B 0,C 180,E1 -9070.136,E2 -9070.136} C_VEL
LIN {X 0,Y 440.409,Z 190.134,A -85,B 0,C 180,E1 -9071.858,E2 -9071.858} C_VEL
LIN {X 0,Y 444.015,Z 213.658,A -85,B 0,C 180,E1 -9072.402,E2 -9072.402} C_VEL
LIN {X 0,Y 443.219,Z 298.627,A -85,B 0,C 180,E1 -9073.8,E2 -9073.8} C_VEL
LIN {X 0,Y 442.738,Z 311.884,A -85,B 0,C 180,E1 -9074.196,E2 -9074.196} C_VEL
LIN {X 0,Y 442.214,Z 324.044,A -85,B 0,C 180,E1 -9074.738,E2 -9074.738} C_VEL
LIN {X 0,Y 441.558,Z 336.316,A -85,B 0,C 180,E1 -9075.482,E2 -9075.482} C_VEL
LIN {X 0,Y 440.863,Z 348.398,A -85,B 0,C 180,E1 -9076.443,E2 -9076.443} C_VEL
LIN {X 0,Y 440.268,Z 359.422,A -85,B 0,C 180,E1 -9077.555,E2 -9077.555} C_VEL
LIN {X 0,Y 439.673,Z 368.605,A -85,B 0,C 180,E1 -9078.708,E2 -9078.708} C_VEL
LIN {X 0,Y 439.133,Z 377.557,A -85,B 0,C 180,E1 -9080.093,E2 -9080.093} C_VEL
LIN {X 0,Y 438.77,Z 384.766,A -85,B 0,C 180,E1 -9081.479,E2 -9081.479} C_VEL
LIN {X 0,Y 438.528,Z 389.632,A -85,B 0,C 180,E1 -9082.633,E2 -9082.633} C_VEL
LIN {X 0,Y 438.345,Z 394.388,A -85,B 0,C 180,E1 -9084.026,E2 -9084.026} C_VEL
LIN {X 0,Y 438.339,Z 397.982,A -85,B 0,C 180,E1 -9085.401,E2 -9085.401} C_VEL
LIN {X 0,Y 438.282,Z 399.847,A -85,B 0,C 180,E1 -9086.322,E2 -9086.322} C_VEL
LIN {X 0,Y 438.341,Z 401.249,A -85,B 0,C 180,E1 -9087.243,E2 -9087.243} C_VEL
LIN {X 0,Y 438.28,Z 402.855,A -85,B 0,C 180,E1 -9089.081,E2 -9089.081} C_VEL
LIN {X 0,Y 438.285,Z 403.072,A -85,B 0,C 180,E1 -9090,E2 -9090} C_VEL
LIN {X 0,Y 438.28,Z 402.854,A -85,B 0,C 180,E1 -9090.918,E2 -9090.918} C_VEL
LIN {X 0,Y 438.341,Z 401.249,A -85,B 0,C 180,E1 -9092.756,E2 -9092.756} C_VEL
LIN {X 0,Y 438.282,Z 399.846,A -85,B 0,C 180,E1 -9093.677,E2 -9093.677} C_VEL
LIN {X 0,Y 438.379,Z 396.904,A -85,B 0,C 180,E1 -9095.058,E2 -9095.058} C_VEL
LIN {X 0,Y 438.448,Z 392.919,A -85,B 0,C 180,E1 -9096.442,E2 -9096.442} C_VEL
LIN {X 0,Y 438.664,Z 386.794,A -85,B 0,C 180,E1 -9098.058,E2 -9098.058} C_VEL
LIN {X 0,Y 438.961,Z 380.103,A -85,B 0,C 180,E1 -9099.445,E2 -9099.445} C_VEL
LIN {X 0,Y 439.411,Z 371.806,A -85,B 0,C 180,E1 -9100.831,E2 -9100.831} C_VEL
LIN {X 0,Y 440.027,Z 363.308,A -85,B 0,C 180,E1 -9101.983,E2 -9101.983} C_VEL
LIN {X 0,Y 440.604,Z 353.447,A -85,B 0,C 180,E1 -9103.073,E2 -9103.073} C_VEL
LIN {X 0,Y 441.241,Z 342.417,A -85,B 0,C 180,E1 -9104.057,E2 -9104.057} C_VEL
LIN {X 0,Y 441.842,Z 331.031,A -85,B 0,C 180,E1 -9104.861,E2 -9104.861} C_VEL
LIN {X 0,Y 442.422,Z 319.351,A -85,B 0,C 180,E1 -9105.489,E2 -9105.489} C_VEL
LIN {X 0,Y 442.993,Z 305.895,A -85,B 0,C 180,E1 -9106,E2 -9106} C_VEL
LIN {X 0,Y 443.329,Z 292.577,A -85,B 0,C 180,E1 -9106.313,E2 -9106.313} C_VEL
LIN {X 0,Y 443.854,Z 212.237,A -85,B 0,C 180,E1 -9107.623,E2 -9107.623} C_VEL
LIN {X 0,Y 440.419,Z 190.093,A -85,B 0,C 180,E1 -9108.143,E2 -9108.143} C_VEL
LIN {X 0,Y 441.438,Z 170.613,A -85,B 0,C 180,E1 -9111.724,E2 -9111.724} C_VEL
LIN {X 0,Y 442.071,Z 157.527,A -85,B 0,C 180,E1 -9114.164,E2 -9114.164} C_VEL
LIN {X 0,Y 439.781,Z 145.612,A -85,B 0,C 180,E1 -9116.58,E2 -9116.58} C_VEL
LIN {X 0,Y 439.411,Z 143.752,A -85,B 0,C 180,E1 -9116.989,E2 -9116.989} C_VEL
LIN {X 0,Y 439.376,Z 143.755,A -85,B 0,C 180,E1 -9120.259,E2 -9120.259} C_VEL
LIN {X 0,Y 439.36,Z 143.757,A -85,B 0,C 180,E1 -9123.717,E2 -9123.717} C_VEL
LIN {X 0,Y 439.367,Z 143.752,A -85,B 0,C 180,E1 -9126.287,E2 -9126.287} C_VEL
LIN {X 0,Y 439.354,Z 143.756,A -85,B 0,C 180,E1 -9129.779,E2 -9129.779} C_VEL
LIN {X 0,Y 439.338,Z 143.756,A -85,B 0,C 180,E1 -9132.621,E2 -9132.621} C_VEL
LIN {X 0,Y 439.391,Z 143.755,A -85,B 0,C 180,E1 -9135.269,E2 -9135.269} C_VEL
LIN {X 0,Y 439.348,Z 143.76,A -85,B 0,C 180,E1 -9139.015,E2 -9139.015} C_VEL
LIN {X 0,Y 439.36,Z 143.754,A -85,B 0,C 180,E1 -9141.608,E2 -9141.608} C_VEL
LIN {X 0,Y 439.387,Z 143.755,A -85,B 0,C 180,E1 -9144.843,E2 -9144.843} C_VEL
LIN {X 0,Y 439.358,Z 143.753,A -85,B 0,C 180,E1 -9148.138,E2 -9148.138} C_VEL
LIN {X 0,Y 439.391,Z 143.749,A -85,B 0,C 180,E1 -9151.606,E2 -9151.606} C_VEL
LIN {X 0,Y 439.357,Z 143.757,A -85,B 0,C 180,E1 -9154.412,E2 -9154.412} C_VEL
LIN {X 0,Y 439.351,Z 143.754,A -85,B 0,C 180,E1 -9157.424,E2 -9157.424} C_VEL
LIN {X 0,Y 439.431,Z 143.749,A -85,B 0,C 180,E1 -9160.663,E2 -9160.663} C_VEL
LIN {X 0,Y 439.406,Z 143.752,A -85,B 0,C 180,E1 -9164.222,E2 -9164.222} C_VEL
LIN {X 0,Y 439.474,Z 143.738,A -85,B 0,C 180,E1 -9167.285,E2 -9167.285} C_VEL
LIN {X 0,Y 439.464,Z 143.741,A -85,B 0,C 180,E1 -9170.798,E2 -9170.798} C_VEL
LIN {X 0,Y 439.546,Z 143.73,A -85,B 0,C 180,E1 -9173.574,E2 -9173.574} C_VEL
LIN {X 0,Y 439.392,Z 143.749,A -85,B 0,C 180,E1 -9175.413,E2 -9175.413} C_VEL
LIN {X 0,Y 439.615,Z 143.726,A -85,B 0,C 180,E1 -9178.168,E2 -9178.168} C_VEL
LIN {X 0,Y 439.658,Z 143.722,A -85,B 0,C 180,E1 -9180,E2 -9180} C_VEL
LIN {X 0,Y 439.593,Z 143.723,A -85,B 0,C 180,E1 -9182.749,E2 -9182.749} C_VEL
LIN {X 0,Y 439.55,Z 143.73,A -85,B 0,C 180,E1 -9186.426,E2 -9186.426} C_VEL
LIN {X 0,Y 439.483,Z 143.739,A -85,B 0,C 180,E1 -9189.202,E2 -9189.202} C_VEL
LIN {X 0,Y 439.455,Z 143.741,A -85,B 0,C 180,E1 -9192.938,E2 -9192.938} C_VEL
LIN {X 0,Y 439.392,Z 143.748,A -85,B 0,C 180,E1 -9196.328,E2 -9196.328} C_VEL
LIN {X 0,Y 439.392,Z 143.753,A -85,B 0,C 180,E1 -9199.627,E2 -9199.627} C_VEL
LIN {X 0,Y 439.353,Z 143.754,A -85,B 0,C 180,E1 -9202.576,E2 -9202.576} C_VEL
LIN {X 0,Y 439.357,Z 143.756,A -85,B 0,C 180,E1 -9205.588,E2 -9205.588} C_VEL
LIN {X 0,Y 439.382,Z 143.751,A -85,B 0,C 180,E1 -9208.676,E2 -9208.676} C_VEL
LIN {X 0,Y 439.358,Z 143.752,A -85,B 0,C 180,E1 -9212.03,E2 -9212.03} C_VEL
LIN {X 0,Y 439.385,Z 143.752,A -85,B 0,C 180,E1 -9215.341,E2 -9215.341} C_VEL
LIN {X 0,Y 439.361,Z 143.756,A -85,B 0,C 180,E1 -9218.597,E2 -9218.597} C_VEL
LIN {X 0,Y 439.36,Z 143.755,A -85,B 0,C 180,E1 -9221.254,E2 -9221.254} C_VEL
LIN {X 0,Y 439.392,Z 143.756,A -85,B 0,C 180,E1 -9224.731,E2 -9224.731} C_VEL
LIN {X 0,Y 439.38,Z 143.75,A -85,B 0,C 180,E1 -9227.795,E2 -9227.795} C_VEL
LIN {X 0,Y 439.354,Z 143.756,A -85,B 0,C 180,E1 -9230.221,E2 -9230.221} C_VEL
LIN {X 0,Y 439.369,Z 143.752,A -85,B 0,C 180,E1 -9233.714,E2 -9233.714} C_VEL
LIN {X 0,Y 439.37,Z 143.752,A -85,B 0,C 180,E1 -9237.055,E2 -9237.055} C_VEL
LIN {X 0,Y 439.371,Z 143.759,A -85,B 0,C 180,E1 -9240.274,E2 -9240.274} C_VEL
LIN {X 0,Y 439.377,Z 143.75,A -85,B 0,C 180,E1 -9243.394,E2 -9243.394} C_VEL
LIN {X 0,Y 439.382,Z 143.753,A -85,B 0,C 180,E1 -9246.43,E2 -9246.43} C_VEL
LIN {X 0,Y 439.438,Z 143.84,A -85,B 0,C 180,E1 -9248.331,E2 -9248.331} C_VEL
LIN {X 0,Y 440.941,Z 151.623,A -85,B 0,C 180,E1 -9250.116,E2 -9250.116} C_VEL
LIN {X 0,Y 440.787,Z 160.305,A -85,B 0,C 180,E1 -9251.941,E2 -9251.941} C_VEL
LIN {X 0,Y 444.349,Z 178.266,A -85,B 0,C 180,E1 -9252.392,E2 -9252.392} C_VEL
LIN {X 0,Y 443.385,Z 267.923,A -85,B 0,C 180,E1 -9253.867,E2 -9253.867} C_VEL
LIN {X 0,Y 443.211,Z 277.666,A -85,B 0,C 180,E1 -9254.147,E2 -9254.147} C_VEL
LIN {X 0,Y 442.383,Z 283.361,A -85,B 0,C 180,E1 -9254.326,E2 -9254.326} C_VEL
LIN {X 0,Y 439.252,Z 292.471,A -85,B 0,C 180,E1 -9254.64,E2 -9254.64} C_VEL
LIN {X 0,Y 436.081,Z 301.277,A -85,B 0,C 180,E1 -9255.06,E2 -9255.06} C_VEL
LIN {X 0,Y 435.192,Z 306.489,A -85,B 0,C 180,E1 -9255.402,E2 -9255.402} C_VEL
LIN {X 0,Y 434.693,Z 317.337,A -85,B 0,C 180,E1 -9256.297,E2 -9256.297} C_VEL
LIN {X 0,Y 433.967,Z 327.847,A -85,B 0,C 180,E1 -9257.372,E2 -9257.372} C_VEL
LIN {X 0,Y 433.347,Z 337.022,A -85,B 0,C 180,E1 -9258.541,E2 -9258.541} C_VEL
LIN {X 0,Y 432.699,Z 345.929,A -85,B 0,C 180,E1 -9259.945,E2 -9259.945} C_VEL
LIN {X 0,Y 432.188,Z 353.098,A -85,B 0,C 180,E1 -9261.349,E2 -9261.349} C_VEL
LIN {X 0,Y 431.891,Z 357.931,A -85,B 0,C 180,E1 -9262.521,E2 -9262.521} C_VEL
LIN {X 0,Y 431.705,Z 362.624,A -85,B 0,C 180,E1 -9263.926,E2 -9263.926} C_VEL
LIN {X 0,Y 431.411,Z 366.223,A -85,B 0,C 180,E1 -9265.328,E2 -9265.328} C_VEL
LIN {X 0,Y 431.439,Z 368.076,A -85,B 0,C 180,E1 -9266.265,E2 -9266.265} C_VEL
LIN {X 0,Y 431.36,Z 369.477,A -85,B 0,C 180,E1 -9267.199,E2 -9267.199} C_VEL
LIN {X 0,Y 431.201,Z 371.088,A -85,B 0,C 180,E1 -9269.067,E2 -9269.067} C_VEL
LIN {X 0,Y 431.199,Z 371.322,A -85,B 0,C 180,E1 -9270,E2 -9270} C_VEL
LIN {X 0,Y 431.201,Z 371.135,A -85,B 0,C 180,E1 -9270.934,E2 -9270.934} C_VEL
LIN {X 0,Y 431.359,Z 369.585,A -85,B 0,C 180,E1 -9272.802,E2 -9272.802} C_VEL
LIN {X 0,Y 431.424,Z 368.233,A -85,B 0,C 180,E1 -9273.737,E2 -9273.737} C_VEL
LIN {X 0,Y 431.469,Z 365.377,A -85,B 0,C 180,E1 -9275.14,E2 -9275.14} C_VEL
LIN {X 0,Y 431.725,Z 361.498,A -85,B 0,C 180,E1 -9276.544,E2 -9276.544} C_VEL
LIN {X 0,Y 431.957,Z 356.496,A -85,B 0,C 180,E1 -9277.95,E2 -9277.95} C_VEL
LIN {X 0,Y 432.445,Z 350.194,A -85,B 0,C 180,E1 -9279.353,E2 -9279.353} C_VEL
LIN {X 0,Y 432.942,Z 342.307,A -85,B 0,C 180,E1 -9280.759,E2 -9280.759} C_VEL
LIN {X 0,Y 433.501,Z 334.263,A -85,B 0,C 180,E1 -9281.93,E2 -9281.93} C_VEL
LIN {X 0,Y 434.235,Z 324.441,A -85,B 0,C 180,E1 -9283.097,E2 -9283.097} C_VEL
LIN {X 0,Y 434.833,Z 313.671,A -85,B 0,C 180,E1 -9284.127,E2 -9284.127} C_VEL
LIN {X 0,Y 435.443,Z 302.569,A -85,B 0,C 180,E1 -9284.966,E2 -9284.966} C_VEL
LIN {X 0,Y 435.972,Z 290.605,A -85,B 0,C 180,E1 -9285.665,E2 -9285.665} C_VEL
LIN {X 0,Y 436.424,Z 277.471,A -85,B 0,C 180,E1 -9286.219,E2 -9286.219} C_VEL
LIN {X 0,Y 436.79,Z 264.247,A -85,B 0,C 180,E1 -9286.565,E2 -9286.565} C_VEL
LIN {X 0,Y 437.497,Z 178.485,A -85,B 0,C 180,E1 -9287.991,E2 -9287.991} C_VEL
LIN {X 0,Y 433.868,Z 160.447,A -85,B 0,C 180,E1 -9288.463,E2 -9288.463} C_VEL
LIN {X 0,Y 433.985,Z 152.957,A -85,B 0,C 180,E1 -9290.072,E2 -9290.072} C_VEL
LIN {X 0,Y 432.34,Z 144.632,A -85,B 0,C 180,E1 -9292.013,E2 -9292.013} C_VEL
LIN {X 0,Y 432.339,Z 144.628,A -85,B 0,C 180,E1 -9295.002,E2 -9295.002} C_VEL
LIN {X 0,Y 432.349,Z 144.63,A -85,B 0,C 180,E1 -9298.126,E2 -9298.126} C_VEL
LIN {X 0,Y 432.323,Z 144.632,A -85,B 0,C 180,E1 -9301.346,E2 -9301.346} C_VEL
LIN {X 0,Y 432.341,Z 144.627,A -85,B 0,C 180,E1 -9304.677,E2 -9304.677} C_VEL
LIN {X 0,Y 432.33,Z 144.629,A -85,B 0,C 180,E1 -9308.151,E2 -9308.151} C_VEL
LIN {X 0,Y 432.321,Z 144.632,A -85,B 0,C 180,E1 -9311.798,E2 -9311.798} C_VEL
LIN {X 0,Y 432.334,Z 144.627,A -85,B 0,C 180,E1 -9314.347,E2 -9314.347} C_VEL
LIN {X 0,Y 432.316,Z 144.634,A -85,B 0,C 180,E1 -9317.016,E2 -9317.016} C_VEL
LIN {X 0,Y 432.308,Z 144.632,A -85,B 0,C 180,E1 -9319.824,E2 -9319.824} C_VEL
LIN {X 0,Y 432.303,Z 144.637,A -85,B 0,C 180,E1 -9323.021,E2 -9323.021} C_VEL
LIN {X 0,Y 432.331,Z 144.628,A -85,B 0,C 180,E1 -9326.002,E2 -9326.002} C_VEL
LIN {X 0,Y 432.342,Z 144.628,A -85,B 0,C 180,E1 -9329.49,E2 -9329.49} C_VEL
LIN {X 0,Y 432.337,Z 144.627,A -85,B 0,C 180,E1 -9331.873,E2 -9331.873} C_VEL
LIN {X 0,Y 432.375,Z 144.623,A -85,B 0,C 180,E1 -9335.539,E2 -9335.539} C_VEL
LIN {X 0,Y 432.347,Z 144.629,A -85,B 0,C 180,E1 -9339.046,E2 -9339.046} C_VEL
LIN {X 0,Y 432.345,Z 144.627,A -85,B 0,C 180,E1 -9342.01,E2 -9342.01} C_VEL
LIN {X 0,Y 432.346,Z 144.629,A -85,B 0,C 180,E1 -9344.925,E2 -9344.925} C_VEL
LIN {X 0,Y 432.456,Z 144.613,A -85,B 0,C 180,E1 -9347.803,E2 -9347.803} C_VEL
LIN {X 0,Y 432.459,Z 144.612,A -85,B 0,C 180,E1 -9351.59,E2 -9351.59} C_VEL
LIN {X 0,Y 432.547,Z 144.606,A -85,B 0,C 180,E1 -9354.405,E2 -9354.405} C_VEL
LIN {X 0,Y 432.592,Z 144.603,A -85,B 0,C 180,E1 -9358.138,E2 -9358.138} C_VEL
LIN {X 0,Y 432.616,Z 144.599,A -85,B 0,C 180,E1 -9360,E2 -9360} C_VEL
LIN {X 0,Y 432.551,Z 144.601,A -85,B 0,C 180,E1 -9362.794,E2 -9362.794} C_VEL
LIN {X 0,Y 432.51,Z 144.607,A -85,B 0,C 180,E1 -9366.531,E2 -9366.531} C_VEL
LIN {X 0,Y 432.414,Z 144.62,A -85,B 0,C 180,E1 -9369.354,E2 -9369.354} C_VEL
LIN {X 0,Y 432.415,Z 144.617,A -85,B 0,C 180,E1 -9372.795,E2 -9372.795} C_VEL
LIN {X 0,Y 432.352,Z 144.625,A -85,B 0,C 180,E1 -9376.453,E2 -9376.453} C_VEL
LIN {X 0,Y 432.31,Z 144.633,A -85,B 0,C 180,E1 -9379.962,E2 -9379.962} C_VEL
LIN {X 0,Y 432.299,Z 144.634,A -85,B 0,C 180,E1 -9382.965,E2 -9382.965} C_VEL
LIN {X 0,Y 432.314,Z 144.631,A -85,B 0,C 180,E1 -9386.036,E2 -9386.036} C_VEL
LIN {X 0,Y 432.312,Z 144.637,A -85,B 0,C 180,E1 -9389.19,E2 -9389.19} C_VEL
LIN {X 0,Y 432.313,Z 144.631,A -85,B 0,C 180,E1 -9392.444,E2 -9392.444} C_VEL
LIN {X 0,Y 432.334,Z 144.628,A -85,B 0,C 180,E1 -9395.818,E2 -9395.818} C_VEL
LIN {X 0,Y 432.328,Z 144.632,A -85,B 0,C 180,E1 -9398.713,E2 -9398.713} C_VEL
LIN {X 0,Y 432.302,Z 144.631,A -85,B 0,C 180,E1 -9401.801,E2 -9401.801} C_VEL
LIN {X 0,Y 432.333,Z 144.63,A -85,B 0,C 180,E1 -9404.348,E2 -9404.348} C_VEL
LIN {X 0,Y 432.302,Z 144.635,A -85,B 0,C 180,E1 -9407.019,E2 -9407.019} C_VEL
LIN {X 0,Y 432.289,Z 144.633,A -85,B 0,C 180,E1 -9409.828,E2 -9409.828} C_VEL
LIN {X 0,Y 432.304,Z 144.633,A -85,B 0,C 180,E1 -9413.022,E2 -9413.022} C_VEL
LIN {X 0,Y 432.333,Z 144.63,A -85,B 0,C 180,E1 -9416.002,E2 -9416.002} C_VEL
LIN {X 0,Y 432.347,Z 144.629,A -85,B 0,C 180,E1 -9419.49,E2 -9419.49} C_VEL
LIN {X 0,Y 432.393,Z 144.709,A -85,B 0,C 180,E1 -9422.797,E2 -9422.797} C_VEL
LIN {X 0,Y 435.116,Z 158.608,A -85,B 0,C 180,E1 -9425.677,E2 -9425.677} C_VEL
LIN {X 0,Y 434.653,Z 169.075,A -85,B 0,C 180,E1 -9427.668,E2 -9427.668} C_VEL
LIN {X 0,Y 433.597,Z 187.329,A -85,B 0,C 180,E1 -9431.084,E2 -9431.084} C_VEL
LIN {X 0,Y 433.478,Z 189.876,A -85,B 0,C 180,E1 -9431.559,E2 -9431.559} C_VEL
LIN {X 0,Y 437.241,Z 214.391,A -85,B 0,C 180,E1 -9432.137,E2 -9432.137} C_VEL
LIN {X 0,Y 436.418,Z 298.38,A -85,B 0,C 180,E1 -9433.541,E2 -9433.541} C_VEL
LIN {X 0,Y 435.927,Z 311.633,A -85,B 0,C 180,E1 -9433.943,E2 -9433.943} C_VEL
LIN {X 0,Y 435.352,Z 323.79,A -85,B 0,C 180,E1 -9434.492,E2 -9434.492} C_VEL
LIN {X 0,Y 434.681,Z 336.061,A -85,B 0,C 180,E1 -9435.247,E2 -9435.247} C_VEL
LIN {X 0,Y 433.99,Z 347.21,A -85,B 0,C 180,E1 -9436.139,E2 -9436.139} C_VEL
LIN {X 0,Y 433.301,Z 358.117,A -85,B 0,C 180,E1 -9437.232,E2 -9437.232} C_VEL
LIN {X 0,Y 432.796,Z 366.667,A -85,B 0,C 180,E1 -9438.288,E2 -9438.288} C_VEL
LIN {X 0,Y 432.24,Z 374.554,A -85,B 0,C 180,E1 -9439.46,E2 -9439.46} C_VEL
LIN {X 0,Y 431.794,Z 382.262,A -85,B 0,C 180,E1 -9440.869,E2 -9440.869} C_VEL
LIN {X 0,Y 431.458,Z 389.373,A -85,B 0,C 180,E1 -9442.512,E2 -9442.512} C_VEL
LIN {X 0,Y 431.316,Z 393.424,A -85,B 0,C 180,E1 -9443.697,E2 -9443.697} C_VEL
LIN {X 0,Y 431.268,Z 397.724,A -85,B 0,C 180,E1 -9445.326,E2 -9445.326} C_VEL
LIN {X 0,Y 431.188,Z 399.588,A -85,B 0,C 180,E1 -9446.261,E2 -9446.261} C_VEL
LIN {X 0,Y 431.237,Z 400.989,A -85,B 0,C 180,E1 -9447.197,E2 -9447.197} C_VEL
LIN {X 0,Y 431.219,Z 401.988,A -85,B 0,C 180,E1 -9448.132,E2 -9448.132} C_VEL
LIN {X 0,Y 431.195,Z 402.596,A -85,B 0,C 180,E1 -9449.066,E2 -9449.066} C_VEL
LIN {X 0,Y 431.197,Z 402.813,A -85,B 0,C 180,E1 -9450,E2 -9450} C_VEL
LIN {X 0,Y 431.195,Z 402.595,A -85,B 0,C 180,E1 -9450.933,E2 -9450.933} C_VEL
LIN {X 0,Y 431.219,Z 401.987,A -85,B 0,C 180,E1 -9451.867,E2 -9451.867} C_VEL
LIN {X 0,Y 431.237,Z 400.989,A -85,B 0,C 180,E1 -9452.802,E2 -9452.802} C_VEL
LIN {X 0,Y 431.188,Z 399.586,A -85,B 0,C 180,E1 -9453.738,E2 -9453.738} C_VEL
LIN {X 0,Y 431.289,Z 396.643,A -85,B 0,C 180,E1 -9455.141,E2 -9455.141} C_VEL
LIN {X 0,Y 431.375,Z 392.658,A -85,B 0,C 180,E1 -9456.548,E2 -9456.548} C_VEL
LIN {X 0,Y 431.593,Z 386.532,A -85,B 0,C 180,E1 -9458.191,E2 -9458.191} C_VEL
LIN {X 0,Y 431.911,Z 379.841,A -85,B 0,C 180,E1 -9459.6,E2 -9459.6} C_VEL
LIN {X 0,Y 432.407,Z 371.543,A -85,B 0,C 180,E1 -9461.009,E2 -9461.009} C_VEL
LIN {X 0,Y 433.045,Z 363.045,A -85,B 0,C 180,E1 -9462.179,E2 -9462.179} C_VEL
LIN {X 0,Y 433.64,Z 353.587,A -85,B 0,C 180,E1 -9463.246,E2 -9463.246} C_VEL
LIN {X 0,Y 434.322,Z 342.153,A -85,B 0,C 180,E1 -9464.286,E2 -9464.286} C_VEL
LIN {X 0,Y 434.956,Z 330.766,A -85,B 0,C 180,E1 -9465.102,E2 -9465.102} C_VEL
LIN {X 0,Y 435.569,Z 319.085,A -85,B 0,C 180,E1 -9465.739,E2 -9465.739} C_VEL
LIN {X 0,Y 436.177,Z 305.626,A -85,B 0,C 180,E1 -9466.257,E2 -9466.257} C_VEL
LIN {X 0,Y 436.52,Z 292.3,A -85,B 0,C 180,E1 -9466.574,E2 -9466.574} C_VEL
LIN {X 0,Y 437.113,Z 213.22,A -85,B 0,C 180,E1 -9467.882,E2 -9467.882} C_VEL
LIN {X 0,Y 433.499,Z 189.86,A -85,B 0,C 180,E1 -9468.437,E2 -9468.437} C_VEL
LIN {X 0,Y 434.49,Z 171.657,A -85,B 0,C 180,E1 -9471.84,E2 -9471.84} C_VEL
LIN {X 0,Y 435.175,Z 159.888,A -85,B 0,C 180,E1 -9474.065,E2 -9474.065} C_VEL
LIN {X 0,Y 434.112,Z 153.185,A -85,B 0,C 180,E1 -9475.423,E2 -9475.423} C_VEL
LIN {X 0,Y 432.375,Z 144.626,A -85,B 0,C 180,E1 -9477.235,E2 -9477.235} C_VEL
LIN {X 0,Y 432.343,Z 144.63,A -85,B 0,C 180,E1 -9480.509,E2 -9480.509} C_VEL
LIN {X 0,Y 432.329,Z 144.63,A -85,B 0,C 180,E1 -9483.997,E2 -9483.997} C_VEL
LIN {X 0,Y 432.316,Z 144.634,A -85,B 0,C 180,E1 -9487.195,E2 -9487.195} C_VEL
LIN {X 0,Y 432.286,Z 144.634,A -85,B 0,C 180,E1 -9490.172,E2 -9490.172} C_VEL
LIN {X 0,Y 432.301,Z 144.636,A -85,B 0,C 180,E1 -9493.061,E2 -9493.061} C_VEL
LIN {X 0,Y 432.327,Z 144.631,A -85,B 0,C 180,E1 -9495.664,E2 -9495.664} C_VEL
LIN {X 0,Y 432.302,Z 144.632,A -85,B 0,C 180,E1 -9498.401,E2 -9498.401} C_VEL
LIN {X 0,Y 432.324,Z 144.629,A -85,B 0,C 180,E1 -9501.849,E2 -9501.849} C_VEL
LIN {X 0,Y 432.319,Z 144.632,A -85,B 0,C 180,E1 -9505.321,E2 -9505.321} C_VEL
LIN {X 0,Y 432.307,Z 144.636,A -85,B 0,C 180,E1 -9508.653,E2 -9508.653} C_VEL
LIN {X 0,Y 432.319,Z 144.629,A -85,B 0,C 180,E1 -9511.872,E2 -9511.872} C_VEL
LIN {X 0,Y 432.344,Z 144.626,A -85,B 0,C 180,E1 -9515.545,E2 -9515.545} C_VEL
LIN {X 0,Y 432.336,Z 144.629,A -85,B 0,C 180,E1 -9519.045,E2 -9519.045} C_VEL
LIN {X 0,Y 432.325,Z 144.631,A -85,B 0,C 180,E1 -9522.009,E2 -9522.009} C_VEL
LIN {X 0,Y 432.338,Z 144.629,A -85,B 0,C 180,E1 -9524.924,E2 -9524.924} C_VEL
LIN {X 0,Y 432.444,Z 144.616,A -85,B 0,C 180,E1 -9527.803,E2 -9527.803} C_VEL
LIN {X 0,Y 432.436,Z 144.616,A -85,B 0,C 180,E1 -9531.589,E2 -9531.589} C_VEL
LIN {X 0,Y 432.539,Z 144.606,A -85,B 0,C 180,E1 -9534.405,E2 -9534.405} C_VEL
LIN {X 0,Y 432.584,Z 144.602,A -85,B 0,C 180,E1 -9538.138,E2 -9538.138} C_VEL
LIN {X 0,Y 432.609,Z 144.6,A -85,B 0,C 180,E1 -9540,E2 -9540} C_VEL
LIN {X 0,Y 432.547,Z 144.601,A -85,B 0,C 180,E1 -9542.794,E2 -9542.794} C_VEL
LIN {X 0,Y 432.561,Z 144.604,A -85,B 0,C 180,E1 -9545.594,E2 -9545.594} C_VEL
LIN {X 0,Y 432.453,Z 144.613,A -85,B 0,C 180,E1 -9548.411,E2 -9548.411} C_VEL
LIN {X 0,Y 432.449,Z 144.615,A -85,B 0,C 180,E1 -9552.197,E2 -9552.197} C_VEL
LIN {X 0,Y 432.379,Z 144.624,A -85,B 0,C 180,E1 -9556.041,E2 -9556.041} C_VEL
LIN {X 0,Y 432.377,Z 144.629,A -85,B 0,C 180,E1 -9559.485,E2 -9559.485} C_VEL
LIN {X 0,Y 432.302,Z 144.635,A -85,B 0,C 180,E1 -9562.965,E2 -9562.965} C_VEL
LIN {X 0,Y 432.31,Z 144.631,A -85,B 0,C 180,E1 -9566.036,E2 -9566.036} C_VEL
LIN {X 0,Y 432.319,Z 144.637,A -85,B 0,C 180,E1 -9569.189,E2 -9569.189} C_VEL
LIN {X 0,Y 432.314,Z 144.631,A -85,B 0,C 180,E1 -9572.444,E2 -9572.444} C_VEL
LIN {X 0,Y 432.33,Z 144.628,A -85,B 0,C 180,E1 -9575.819,E2 -9575.819} C_VEL
LIN {X 0,Y 432.323,Z 144.634,A -85,B 0,C 180,E1 -9578.713,E2 -9578.713} C_VEL
LIN {X 0,Y 432.302,Z 144.631,A -85,B 0,C 180,E1 -9581.801,E2 -9581.801} C_VEL
LIN {X 0,Y 432.328,Z 144.631,A -85,B 0,C 180,E1 -9584.348,E2 -9584.348} C_VEL
LIN {X 0,Y 432.312,Z 144.633,A -85,B 0,C 180,E1 -9587.017,E2 -9587.017} C_VEL
LIN {X 0,Y 432.309,Z 144.631,A -85,B 0,C 180,E1 -9589.825,E2 -9589.825} C_VEL
LIN {X 0,Y 432.301,Z 144.633,A -85,B 0,C 180,E1 -9593.023,E2 -9593.023} C_VEL
LIN {X 0,Y 432.357,Z 144.627,A -85,B 0,C 180,E1 -9595.998,E2 -9595.998} C_VEL
LIN {X 0,Y 432.344,Z 144.626,A -85,B 0,C 180,E1 -9599.491,E2 -9599.491} C_VEL
LIN {X 0,Y 432.339,Z 144.63,A -85,B 0,C 180,E1 -9601.875,E2 -9601.875} C_VEL
LIN {X 0,Y 432.376,Z 144.623,A -85,B 0,C 180,E1 -9605.54,E2 -9605.54} C_VEL
LIN {X 0,Y 432.367,Z 144.716,A -85,B 0,C 180,E1 -9608.11,E2 -9608.11} C_VEL
LIN {X 0,Y 434.016,Z 153.386,A -85,B 0,C 180,E1 -9610.121,E2 -9610.121} C_VEL
LIN {X 0,Y 433.854,Z 160.455,A -85,B 0,C 180,E1 -9611.637,E2 -9611.637} C_VEL
LIN {X 0,Y 437.586,Z 179.315,A -85,B 0,C 180,E1 -9612.123,E2 -9612.123} C_VEL
LIN {X 0,Y 436.647,Z 266.998,A -85,B 0,C 180,E1 -9613.581,E2 -9613.581} C_VEL
LIN {X 0,Y 436.382,Z 279.756,A -85,B 0,C 180,E1 -9613.961,E2 -9613.961} C_VEL
LIN {X 0,Y 435.847,Z 292.196,A -85,B 0,C 180,E1 -9614.511,E2 -9614.511} C_VEL
LIN {X 0,Y 435.242,Z 304.686,A -85,B 0,C 180,E1 -9615.268,E2 -9615.268} C_VEL
LIN {X 0,Y 435.192,Z 306.489,A -85,B 0,C 180,E1 -9615.402,E2 -9615.402} C_VEL
LIN {X 0,Y 434.299,Z 311.683,A -85,B 0,C 180,E1 -9615.779,E2 -9615.779} C_VEL
LIN {X 0,Y 431.047,Z 319.829,A -85,B 0,C 180,E1 -9616.406,E2 -9616.406} C_VEL
LIN {X 0,Y 427.741,Z 327.469,A -85,B 0,C 180,E1 -9617.115,E2 -9617.115} C_VEL
LIN {X 0,Y 426.75,Z 331.844,A -85,B 0,C 180,E1 -9617.618,E2 -9617.618} C_VEL
LIN {X 0,Y 426.17,Z 340.499,A -85,B 0,C 180,E1 -9618.828,E2 -9618.828} C_VEL
LIN {X 0,Y 425.556,Z 348.746,A -85,B 0,C 180,E1 -9620.255,E2 -9620.255} C_VEL
LIN {X 0,Y 425.091,Z 354.389,A -85,B 0,C 180,E1 -9621.443,E2 -9621.443} C_VEL
LIN {X 0,Y 424.727,Z 360.764,A -85,B 0,C 180,E1 -9623.135,E2 -9623.135} C_VEL
LIN {X 0,Y 424.417,Z 365.422,A -85,B 0,C 180,E1 -9624.775,E2 -9624.775} C_VEL
LIN {X 0,Y 424.344,Z 368.337,A -85,B 0,C 180,E1 -9626.202,E2 -9626.202} C_VEL
LIN {X 0,Y 424.295,Z 369.735,A -85,B 0,C 180,E1 -9627.152,E2 -9627.152} C_VEL
LIN {X 0,Y 424.119,Z 371.347,A -85,B 0,C 180,E1 -9629.051,E2 -9629.051} C_VEL
LIN {X 0,Y 424.115,Z 371.581,A -85,B 0,C 180,E1 -9630,E2 -9630} C_VEL
LIN {X 0,Y 424.119,Z 371.394,A -85,B 0,C 180,E1 -9630.95,E2 -9630.95} C_VEL
LIN {X 0,Y 424.293,Z 369.843,A -85,B 0,C 180,E1 -9632.849,E2 -9632.849} C_VEL
LIN {X 0,Y 424.33,Z 368.492,A -85,B 0,C 180,E1 -9633.799,E2 -9633.799} C_VEL
LIN {X 0,Y 424.416,Z 365.635,A -85,B 0,C 180,E1 -9635.226,E2 -9635.226} C_VEL
LIN {X 0,Y 424.653,Z 361.367,A -85,B 0,C 180,E1 -9636.782,E2 -9636.782} C_VEL
LIN {X 0,Y 424.931,Z 356.754,A -85,B 0,C 180,E1 -9638.082,E2 -9638.082} C_VEL
LIN {X 0,Y 425.426,Z 350.452,A -85,B 0,C 180,E1 -9639.509,E2 -9639.509} C_VEL
LIN {X 0,Y 425.984,Z 342.563,A -85,B 0,C 180,E1 -9640.937,E2 -9640.937} C_VEL
LIN {X 0,Y 426.551,Z 334.519,A -85,B 0,C 180,E1 -9642.127,E2 -9642.127} C_VEL
LIN {X 0,Y 427.347,Z 324.695,A -85,B 0,C 180,E1 -9643.311,E2 -9643.311} C_VEL
LIN {X 0,Y 427.968,Z 313.798,A -85,B 0,C 180,E1 -9644.37,E2 -9644.37} C_VEL
LIN {X 0,Y 428.594,Z 302.821,A -85,B 0,C 180,E1 -9645.211,E2 -9645.211} C_VEL
LIN {X 0,Y 429.151,Z 290.856,A -85,B 0,C 180,E1 -9645.921,E2 -9645.921} C_VEL
LIN {X 0,Y 429.629,Z 278.596,A -85,B 0,C 180,E1 -9646.452,E2 -9646.452} C_VEL
LIN {X 0,Y 429.993,Z 265.987,A -85,B 0,C 180,E1 -9646.804,E2 -9646.804} C_VEL
LIN {X 0,Y 430.804,Z 179.55,A -85,B 0,C 180,E1 -9648.265,E2 -9648.265} C_VEL
LIN {X 0,Y 426.95,Z 160.694,A -85,B 0,C 180,E1 -9648.773,E2 -9648.773} C_VEL
LIN {X 0,Y 427.086,Z 154.654,A -85,B 0,C 180,E1 -9650.085,E2 -9650.085} C_VEL
LIN {X 0,Y 425.295,Z 145.51,A -85,B 0,C 180,E1 -9652.27,E2 -9652.27} C_VEL
LIN {X 0,Y 425.321,Z 145.503,A -85,B 0,C 180,E1 -9654.657,E2 -9654.657} C_VEL
LIN {X 0,Y 425.274,Z 145.511,A -85,B 0,C 180,E1 -9657.563,E2 -9657.563} C_VEL
LIN {X 0,Y 425.292,Z 145.505,A -85,B 0,C 180,E1 -9660.761,E2 -9660.761} C_VEL
LIN {X 0,Y 425.313,Z 145.503,A -85,B 0,C 180,E1 -9664.288,E2 -9664.288} C_VEL
LIN {X 0,Y 425.276,Z 145.512,A -85,B 0,C 180,E1 -9667.694,E2 -9667.694} C_VEL
LIN {X 0,Y 425.247,Z 145.51,A -85,B 0,C 180,E1 -9670.515,E2 -9670.515} C_VEL
LIN {X 0,Y 425.256,Z 145.516,A -85,B 0,C 180,E1 -9673.35,E2 -9673.35} C_VEL
LIN {X 0,Y 425.26,Z 145.509,A -85,B 0,C 180,E1 -9676.044,E2 -9676.044} C_VEL
LIN {X 0,Y 425.258,Z 145.51,A -85,B 0,C 180,E1 -9678.619,E2 -9678.619} C_VEL
LIN {X 0,Y 425.283,Z 145.512,A -85,B 0,C 180,E1 -9681.099,E2 -9681.099} C_VEL
LIN {X 0,Y 425.294,Z 145.507,A -85,B 0,C 180,E1 -9684.663,E2 -9684.663} C_VEL
LIN {X 0,Y 425.259,Z 145.509,A -85,B 0,C 180,E1 -9688.072,E2 -9688.072} C_VEL
LIN {X 0,Y 425.303,Z 145.505,A -85,B 0,C 180,E1 -9691.366,E2 -9691.366} C_VEL
LIN {X 0,Y 425.268,Z 145.512,A -85,B 0,C 180,E1 -9694.553,E2 -9694.553} C_VEL
LIN {X 0,Y 425.302,Z 145.51,A -85,B 0,C 180,E1 -9696.634,E2 -9696.634} C_VEL
LIN {X 0,Y 425.326,Z 145.504,A -85,B 0,C 180,E1 -9700.365,E2 -9700.365} C_VEL
LIN {X 0,Y 425.32,Z 145.501,A -85,B 0,C 180,E1 -9703.685,E2 -9703.685} C_VEL
LIN {X 0,Y 425.391,Z 145.493,A -85,B 0,C 180,E1 -9707.097,E2 -9707.097} C_VEL
LIN {X 0,Y 425.391,Z 145.498,A -85,B 0,C 180,E1 -9710.49,E2 -9710.49} C_VEL
LIN {X 0,Y 425.472,Z 145.482,A -85,B 0,C 180,E1 -9713.36,E2 -9713.36} C_VEL
LIN {X 0,Y 425.339,Z 145.499,A -85,B 0,C 180,E1 -9715.261,E2 -9715.261} C_VEL
LIN {X 0,Y 425.561,Z 145.479,A -85,B 0,C 180,E1 -9718.107,E2 -9718.107} C_VEL
LIN {X 0,Y 425.568,Z 145.477,A -85,B 0,C 180,E1 -9720,E2 -9720} C_VEL
LIN {X 0,Y 425.507,Z 145.478,A -85,B 0,C 180,E1 -9722.84,E2 -9722.84} C_VEL
LIN {X 0,Y 425.471,Z 145.483,A -85,B 0,C 180,E1 -9726.64,E2 -9726.64} C_VEL
LIN {X 0,Y 425.375,Z 145.498,A -85,B 0,C 180,E1 -9729.51,E2 -9729.51} C_VEL
LIN {X 0,Y 425.381,Z 145.494,A -85,B 0,C 180,E1 -9732.898,E2 -9732.898} C_VEL
LIN {X 0,Y 425.31,Z 145.502,A -85,B 0,C 180,E1 -9736.582,E2 -9736.582} C_VEL
LIN {X 0,Y 425.293,Z 145.511,A -85,B 0,C 180,E1 -9739.623,E2 -9739.623} C_VEL
LIN {X 0,Y 425.282,Z 145.506,A -85,B 0,C 180,E1 -9742.339,E2 -9742.339} C_VEL
LIN {X 0,Y 425.256,Z 145.515,A -85,B 0,C 180,E1 -9745.448,E2 -9745.448} C_VEL
LIN {X 0,Y 425.293,Z 145.507,A -85,B 0,C 180,E1 -9748.857,E2 -9748.857} C_VEL
LIN {X 0,Y 425.25,Z 145.51,A -85,B 0,C 180,E1 -9751.928,E2 -9751.928} C_VEL
LIN {X 0,Y 425.293,Z 145.509,A -85,B 0,C 180,E1 -9755.337,E2 -9755.337} C_VEL
LIN {X 0,Y 425.282,Z 145.513,A -85,B 0,C 180,E1 -9758.901,E2 -9758.901} C_VEL
LIN {X 0,Y 425.264,Z 145.508,A -85,B 0,C 180,E1 -9761.954,E2 -9761.954} C_VEL
LIN {X 0,Y 425.284,Z 145.508,A -85,B 0,C 180,E1 -9765.283,E2 -9765.283} C_VEL
LIN {X 0,Y 425.247,Z 145.517,A -85,B 0,C 180,E1 -9768.618,E2 -9768.618} C_VEL
LIN {X 0,Y 425.281,Z 145.508,A -85,B 0,C 180,E1 -9771.099,E2 -9771.099} C_VEL
LIN {X 0,Y 425.295,Z 145.51,A -85,B 0,C 180,E1 -9774.664,E2 -9774.664} C_VEL
LIN {X 0,Y 425.264,Z 145.511,A -85,B 0,C 180,E1 -9778.073,E2 -9778.073} C_VEL
LIN {X 0,Y 425.306,Z 145.507,A -85,B 0,C 180,E1 -9781.366,E2 -9781.366} C_VEL
LIN {X 0,Y 425.343,Z 145.544,A -85,B 0,C 180,E1 -9782.532,E2 -9782.532} C_VEL
LIN {X 0,Y 428.12,Z 159.655,A -85,B 0,C 180,E1 -9785.512,E2 -9785.512} C_VEL
LIN {X 0,Y 427.925,Z 166.704,A -85,B 0,C 180,E1 -9786.884,E2 -9786.884} C_VEL
LIN {X 0,Y 426.77,Z 185.766,A -85,B 0,C 180,E1 -9790.52,E2 -9790.52} C_VEL
LIN {X 0,Y 426.541,Z 189.593,A -85,B 0,C 180,E1 -9791.244,E2 -9791.244} C_VEL
LIN {X 0,Y 430.5,Z 215.72,A -85,B 0,C 180,E1 -9791.875,E2 -9791.875} C_VEL
LIN {X 0,Y 429.631,Z 298.134,A -85,B 0,C 180,E1 -9793.273,E2 -9793.273} C_VEL
LIN {X 0,Y 429.11,Z 311.382,A -85,B 0,C 180,E1 -9793.681,E2 -9793.681} C_VEL
LIN {X 0,Y 428.447,Z 324.657,A -85,B 0,C 180,E1 -9794.296,E2 -9794.296} C_VEL
LIN {X 0,Y 427.787,Z 335.805,A -85,B 0,C 180,E1 -9795.004,E2 -9795.004} C_VEL
LIN {X 0,Y 427.045,Z 347.232,A -85,B 0,C 180,E1 -9795.935,E2 -9795.935} C_VEL
LIN {X 0,Y 426.351,Z 357.859,A -85,B 0,C 180,E1 -9797.021,E2 -9797.021} C_VEL
LIN {X 0,Y 425.804,Z 366.408,A -85,B 0,C 180,E1 -9798.093,E2 -9798.093} C_VEL
LIN {X 0,Y 425.224,Z 374.295,A -85,B 0,C 180,E1 -9799.284,E2 -9799.284} C_VEL
LIN {X 0,Y 424.748,Z 382.003,A -85,B 0,C 180,E1 -9800.716,E2 -9800.716} C_VEL
LIN {X 0,Y 424.494,Z 387.288,A -85,B 0,C 180,E1 -9801.91,E2 -9801.91} C_VEL
LIN {X 0,Y 424.256,Z 392.41,A -85,B 0,C 180,E1 -9803.341,E2 -9803.341} C_VEL
LIN {X 0,Y 424.196,Z 396.391,A -85,B 0,C 180,E1 -9804.771,E2 -9804.771} C_VEL
LIN {X 0,Y 424.099,Z 399.329,A -85,B 0,C 180,E1 -9806.199,E2 -9806.199} C_VEL
LIN {X 0,Y 424.134,Z 400.73,A -85,B 0,C 180,E1 -9807.15,E2 -9807.15} C_VEL
LIN {X 0,Y 424.143,Z 401.729,A -85,B 0,C 180,E1 -9808.1,E2 -9808.1} C_VEL
LIN {X 0,Y 424.113,Z 402.338,A -85,B 0,C 180,E1 -9809.05,E2 -9809.05} C_VEL
LIN {X 0,Y 424.113,Z 402.554,A -85,B 0,C 180,E1 -9810,E2 -9810} C_VEL
LIN {X 0,Y 424.143,Z 401.728,A -85,B 0,C 180,E1 -9811.899,E2 -9811.899} C_VEL
LIN {X 0,Y 424.134,Z 400.729,A -85,B 0,C 180,E1 -9812.849,E2 -9812.849} C_VEL
LIN {X 0,Y 424.099,Z 399.326,A -85,B 0,C 180,E1 -9813.8,E2 -9813.8} C_VEL
LIN {X 0,Y 424.201,Z 396.383,A -85,B 0,C 180,E1 -9815.228,E2 -9815.228} C_VEL
LIN {X 0,Y 424.299,Z 392.397,A -85,B 0,C 180,E1 -9816.658,E2 -9816.658} C_VEL
LIN {X 0,Y 424.526,Z 386.27,A -85,B 0,C 180,E1 -9818.328,E2 -9818.328} C_VEL
LIN {X 0,Y 424.885,Z 379.579,A -85,B 0,C 180,E1 -9819.761,E2 -9819.761} C_VEL
LIN {X 0,Y 425.423,Z 371.281,A -85,B 0,C 180,E1 -9821.192,E2 -9821.192} C_VEL
LIN {X 0,Y 426.061,Z 362.781,A -85,B 0,C 180,E1 -9822.382,E2 -9822.382} C_VEL
LIN {X 0,Y 426.736,Z 352.941,A -85,B 0,C 180,E1 -9823.504,E2 -9823.504} C_VEL
LIN {X 0,Y 427.414,Z 341.889,A -85,B 0,C 180,E1 -9824.522,E2 -9824.522} C_VEL
LIN {X 0,Y 428.112,Z 330.503,A -85,B 0,C 180,E1 -9825.349,E2 -9825.349} C_VEL
LIN {X 0,Y 428.734,Z 318.818,A -85,B 0,C 180,E1 -9825.997,E2 -9825.997} C_VEL
LIN {X 0,Y 429.37,Z 305.358,A -85,B 0,C 180,E1 -9826.522,E2 -9826.522} C_VEL
LIN {X 0,Y 429.721,Z 292.023,A -85,B 0,C 180,E1 -9826.844,E2 -9826.844} C_VEL
LIN {X 0,Y 430.381,Z 214.234,A -85,B 0,C 180,E1 -9828.149,E2 -9828.149} C_VEL
LIN {X 0,Y 426.531,Z 189.599,A -85,B 0,C 180,E1 -9828.748,E2 -9828.748} C_VEL
LIN {X 0,Y 427.53,Z 172.698,A -85,B 0,C 180,E1 -9831.96,E2 -9831.96} C_VEL
LIN {X 0,Y 428.244,Z 160.934,A -85,B 0,C 180,E1 -9834.221,E2 -9834.221} C_VEL
LIN {X 0,Y 426.331,Z 150.354,A -85,B 0,C 180,E1 -9836.428,E2 -9836.428} C_VEL
LIN {X 0,Y 425.325,Z 145.503,A -85,B 0,C 180,E1 -9837.468,E2 -9837.468} C_VEL
LIN {X 0,Y 425.285,Z 145.51,A -85,B 0,C 180,E1 -9840.815,E2 -9840.815} C_VEL
LIN {X 0,Y 425.288,Z 145.506,A -85,B 0,C 180,E1 -9844.283,E2 -9844.283} C_VEL
LIN {X 0,Y 425.271,Z 145.511,A -85,B 0,C 180,E1 -9847.694,E2 -9847.694} C_VEL
LIN {X 0,Y 425.241,Z 145.511,A -85,B 0,C 180,E1 -9850.514,E2 -9850.514} C_VEL
LIN {X 0,Y 425.244,Z 145.517,A -85,B 0,C 180,E1 -9853.349,E2 -9853.349} C_VEL
LIN {X 0,Y 425.251,Z 145.51,A -85,B 0,C 180,E1 -9856.043,E2 -9856.043} C_VEL
LIN {X 0,Y 425.247,Z 145.513,A -85,B 0,C 180,E1 -9859.483,E2 -9859.483} C_VEL
LIN {X 0,Y 425.269,Z 145.509,A -85,B 0,C 180,E1 -9862.488,E2 -9862.488} C_VEL
LIN {X 0,Y 425.278,Z 145.507,A -85,B 0,C 180,E1 -9865.815,E2 -9865.815} C_VEL
LIN {X 0,Y 425.28,Z 145.509,A -85,B 0,C 180,E1 -9869.239,E2 -9869.239} C_VEL
LIN {X 0,Y 425.242,Z 145.515,A -85,B 0,C 180,E1 -9872.435,E2 -9872.435} C_VEL
LIN {X 0,Y 425.314,Z 145.502,A -85,B 0,C 180,E1 -9875.6,E2 -9875.6} C_VEL
LIN {X 0,Y 425.28,Z 145.512,A -85,B 0,C 180,E1 -9878.681,E2 -9878.681} C_VEL
LIN {X 0,Y 425.295,Z 145.505,A -85,B 0,C 180,E1 -9881.701,E2 -9881.701} C_VEL
LIN {X 0,Y 425.291,Z 145.509,A -85,B 0,C 180,E1 -9884.669,E2 -9884.669} C_VEL
LIN {X 0,Y 425.399,Z 145.492,A -85,B 0,C 180,E1 -9887.598,E2 -9887.598} C_VEL
LIN {X 0,Y 425.384,Z 145.494,A -85,B 0,C 180,E1 -9891.449,E2 -9891.449} C_VEL
LIN {X 0,Y 425.497,Z 145.484,A -85,B 0,C 180,E1 -9894.313,E2 -9894.313} C_VEL
LIN {X 0,Y 425.553,Z 145.479,A -85,B 0,C 180,E1 -9898.107,E2 -9898.107} C_VEL
LIN {X 0,Y 425.562,Z 145.478,A -85,B 0,C 180,E1 -9900,E2 -9900} C_VEL
LIN {X 0,Y 425.502,Z 145.479,A -85,B 0,C 180,E1 -9902.84,E2 -9902.84} C_VEL
LIN {X 0,Y 425.467,Z 145.483,A -85,B 0,C 180,E1 -9906.462,E2 -9906.462} C_VEL
LIN {X 0,Y 425.386,Z 145.498,A -85,B 0,C 180,E1 -9909.51,E2 -9909.51} C_VEL
LIN {X 0,Y 425.384,Z 145.494,A -85,B 0,C 180,E1 -9912.904,E2 -9912.904} C_VEL
LIN {X 0,Y 425.308,Z 145.503,A -85,B 0,C 180,E1 -9916.585,E2 -9916.585} C_VEL
LIN {X 0,Y 425.319,Z 145.506,A -85,B 0,C 180,E1 -9919.636,E2 -9919.636} C_VEL
LIN {X 0,Y 425.278,Z 145.506,A -85,B 0,C 180,E1 -9922.339,E2 -9922.339} C_VEL
LIN {X 0,Y 425.251,Z 145.515,A -85,B 0,C 180,E1 -9925.448,E2 -9925.448} C_VEL
LIN {X 0,Y 425.3,Z 145.507,A -85,B 0,C 180,E1 -9928.861,E2 -9928.861} C_VEL
LIN {X 0,Y 425.255,Z 145.51,A -85,B 0,C 180,E1 -9931.928,E2 -9931.928} C_VEL
LIN {X 0,Y 425.289,Z 145.508,A -85,B 0,C 180,E1 -9935.337,E2 -9935.337} C_VEL
LIN {X 0,Y 425.278,Z 145.514,A -85,B 0,C 180,E1 -9938.901,E2 -9938.901} C_VEL
LIN {X 0,Y 425.263,Z 145.509,A -85,B 0,C 180,E1 -9941.956,E2 -9941.956} C_VEL
LIN {X 0,Y 425.28,Z 145.508,A -85,B 0,C 180,E1 -9945.284,E2 -9945.284} C_VEL
LIN {X 0,Y 425.261,Z 145.516,A -85,B 0,C 180,E1 -9948.621,E2 -9948.621} C_VEL
LIN {X 0,Y 425.277,Z 145.508,A -85,B 0,C 180,E1 -9951.1,E2 -9951.1} C_VEL
LIN {X 0,Y 425.296,Z 145.509,A -85,B 0,C 180,E1 -9954.665,E2 -9954.665} C_VEL
LIN {X 0,Y 425.263,Z 145.512,A -85,B 0,C 180,E1 -9958.074,E2 -9958.074} C_VEL
LIN {X 0,Y 425.304,Z 145.503,A -85,B 0,C 180,E1 -9961.367,E2 -9961.367} C_VEL
LIN {X 0,Y 425.269,Z 145.51,A -85,B 0,C 180,E1 -9964.554,E2 -9964.554} C_VEL
LIN {X 0,Y 425.283,Z 145.508,A -85,B 0,C 180,E1 -9966.634,E2 -9966.634} C_VEL
LIN {X 0,Y 425.335,Z 145.665,A -85,B 0,C 180,E1 -9967.897,E2 -9967.897} C_VEL
LIN {X 0,Y 427.067,Z 154.285,A -85,B 0,C 180,E1 -9969.931,E2 -9969.931} C_VEL
LIN {X 0,Y 426.954,Z 160.689,A -85,B 0,C 180,E1 -9971.325,E2 -9971.325} C_VEL
LIN {X 0,Y 430.843,Z 180.035,A -85,B 0,C 180,E1 -9971.841,E2 -9971.841} C_VEL
LIN {X 0,Y 429.845,Z 267.278,A -85,B 0,C 180,E1 -9973.313,E2 -9973.313} C_VEL
LIN {X 0,Y 429.569,Z 280.026,A -85,B 0,C 180,E1 -9973.7,E2 -9973.7} C_VEL
LIN {X 0,Y 429.032,Z 292.463,A -85,B 0,C 180,E1 -9974.258,E2 -9974.258} C_VEL
LIN {X 0,Y 428.383,Z 304.951,A -85,B 0,C 180,E1 -9975.026,E2 -9975.026} C_VEL
LIN {X 0,Y 427.843,Z 315.995,A -85,B 0,C 180,E1 -9975.922,E2 -9975.922} C_VEL
LIN {X 0,Y 427.225,Z 325.985,A -85,B 0,C 180,E1 -9976.928,E2 -9976.928} C_VEL
LIN {X 0,Y 426.75,Z 331.844,A -85,B 0,C 180,E1 -9977.618,E2 -9977.618} C_VEL
LIN {X 0,Y 425.771,Z 336.129,A -85,B 0,C 180,E1 -9978.151,E2 -9978.151} C_VEL
LIN {X 0,Y 422.468,Z 342.72,A -85,B 0,C 180,E1 -9979.049,E2 -9979.049} C_VEL
LIN {X 0,Y 419.208,Z 348.674,A -85,B 0,C 180,E1 -9980.034,E2 -9980.034} C_VEL
LIN {X 0,Y 418.307,Z 351.96,A -85,B 0,C 180,E1 -9980.695,E2 -9980.695} C_VEL
LIN {X 0,Y 417.798,Z 358.453,A -85,B 0,C 180,E1 -9982.267,E2 -9982.267} C_VEL
LIN {X 0,Y 417.587,Z 363.145,A -85,B 0,C 180,E1 -9983.72,E2 -9983.72} C_VEL
LIN {X 0,Y 417.274,Z 366.743,A -85,B 0,C 180,E1 -9985.17,E2 -9985.17} C_VEL
LIN {X 0,Y 417.252,Z 368.597,A -85,B 0,C 180,E1 -9986.137,E2 -9986.137} C_VEL
LIN {X 0,Y 417.23,Z 369.994,A -85,B 0,C 180,E1 -9987.104,E2 -9987.104} C_VEL
LIN {X 0,Y 417.04,Z 371.606,A -85,B 0,C 180,E1 -9989.035,E2 -9989.035} C_VEL
LIN {X 0,Y 417.033,Z 371.839,A -85,B 0,C 180,E1 -9990.001,E2 -9990.001} C_VEL
LIN {X 0,Y 417.04,Z 371.652,A -85,B 0,C 180,E1 -9990.966,E2 -9990.966} C_VEL
LIN {X 0,Y 417.228,Z 370.101,A -85,B 0,C 180,E1 -9992.897,E2 -9992.897} C_VEL
LIN {X 0,Y 417.238,Z 368.75,A -85,B 0,C 180,E1 -9993.864,E2 -9993.864} C_VEL
LIN {X 0,Y 417.366,Z 365.892,A -85,B 0,C 180,E1 -9995.314,E2 -9995.314} C_VEL
LIN {X 0,Y 417.604,Z 361.872,A -85,B 0,C 180,E1 -9996.815,E2 -9996.815} C_VEL
LIN {X 0,Y 417.901,Z 357.011,A -85,B 0,C 180,E1 -9998.219,E2 -9998.219} C_VEL
LIN {X 0,Y 418.427,Z 350.709,A -85,B 0,C 180,E1 -9999.67,E2 -9999.67} C_VEL
LIN {X 0,Y 419.033,Z 342.818,A -85,B 0,C 180,E1 -10001.121,E2 -10001.121} C_VEL
LIN {X 0,Y 419.615,Z 334.775,A -85,B 0,C 180,E1 -10002.331,E2 -10002.331} C_VEL
LIN {X 0,Y 420.46,Z 324.95,A -85,B 0,C 180,E1 -10003.534,E2 -10003.534} C_VEL
LIN {X 0,Y 421.038,Z 315.289,A -85,B 0,C 180,E1 -10004.5,E2 -10004.5} C_VEL
LIN {X 0,Y 421.651,Z 304.832,A -85,B 0,C 180,E1 -10005.344,E2 -10005.344} C_VEL
LIN {X 0,Y 422.297,Z 293.357,A -85,B 0,C 180,E1 -10006.062,E2 -10006.062} C_VEL
LIN {X 0,Y 422.808,Z 280.382,A -85,B 0,C 180,E1 -10006.663,E2 -10006.663} C_VEL
LIN {X 0,Y 423.163,Z 267.686,A -85,B 0,C 180,E1 -10007.052,E2 -10007.052} C_VEL
LIN {X 0,Y 424.015,Z 180.141,A -85,B 0,C 180,E1 -10008.562,E2 -10008.562} C_VEL
LIN {X 0,Y 420.07,Z 160.877,A -85,B 0,C 180,E1 -10009.106,E2 -10009.106} C_VEL
LIN {X 0,Y 420.195,Z 156.921,A -85,B 0,C 180,E1 -10009.976,E2 -10009.976} C_VEL
LIN {X 0,Y 418.581,Z 148.122,A -85,B 0,C 180,E1 -10012.061,E2 -10012.061} C_VEL
LIN {X 0,Y 418.254,Z 146.384,A -85,B 0,C 180,E1 -10012.542,E2 -10012.542} C_VEL
LIN {X 0,Y 418.238,Z 146.391,A -85,B 0,C 180,E1 -10015.906,E2 -10015.906} C_VEL
LIN {X 0,Y 418.263,Z 146.381,A -85,B 0,C 180,E1 -10019.162,E2 -10019.162} C_VEL
LIN {X 0,Y 418.259,Z 146.381,A -85,B 0,C 180,E1 -10022.844,E2 -10022.844} C_VEL
LIN {X 0,Y 418.245,Z 146.384,A -85,B 0,C 180,E1 -10026.237,E2 -10026.237} C_VEL
LIN {X 0,Y 418.201,Z 146.393,A -85,B 0,C 180,E1 -10029.688,E2 -10029.688} C_VEL
LIN {X 0,Y 418.222,Z 146.386,A -85,B 0,C 180,E1 -10032.32,E2 -10032.32} C_VEL
LIN {X 0,Y 418.236,Z 146.388,A -85,B 0,C 180,E1 -10035.108,E2 -10035.108} C_VEL
LIN {X 0,Y 418.232,Z 146.386,A -85,B 0,C 180,E1 -10037.765,E2 -10037.765} C_VEL
LIN {X 0,Y 418.239,Z 146.386,A -85,B 0,C 180,E1 -10041.556,E2 -10041.556} C_VEL
LIN {X 0,Y 418.249,Z 146.388,A -85,B 0,C 180,E1 -10045.158,E2 -10045.158} C_VEL
LIN {X 0,Y 418.241,Z 146.385,A -85,B 0,C 180,E1 -10047.471,E2 -10047.471} C_VEL
LIN {X 0,Y 418.26,Z 146.388,A -85,B 0,C 180,E1 -10050.897,E2 -10050.897} C_VEL
LIN {X 0,Y 418.232,Z 146.385,A -85,B 0,C 180,E1 -10054.093,E2 -10054.093} C_VEL
LIN {X 0,Y 418.236,Z 146.385,A -85,B 0,C 180,E1 -10057.264,E2 -10057.264} C_VEL
LIN {X 0,Y 418.281,Z 146.382,A -85,B 0,C 180,E1 -10060.364,E2 -10060.364} C_VEL
LIN {X 0,Y 418.277,Z 146.379,A -85,B 0,C 180,E1 -10063.403,E2 -10063.403} C_VEL
LIN {X 0,Y 418.344,Z 146.372,A -85,B 0,C 180,E1 -10067,E2 -10067} C_VEL
LIN {X 0,Y 418.332,Z 146.379,A -85,B 0,C 180,E1 -10070.328,E2 -10070.328} C_VEL
LIN {X 0,Y 418.437,Z 146.359,A -85,B 0,C 180,E1 -10073.248,E2 -10073.248} C_VEL
LIN {X 0,Y 418.31,Z 146.374,A -85,B 0,C 180,E1 -10075.181,E2 -10075.181} C_VEL
LIN {X 0,Y 418.53,Z 146.354,A -85,B 0,C 180,E1 -10078.075,E2 -10078.075} C_VEL
LIN {X 0,Y 418.403,Z 146.363,A -85,B 0,C 180,E1 -10080.962,E2 -10080.962} C_VEL
LIN {X 0,Y 418.463,Z 146.355,A -85,B 0,C 180,E1 -10082.888,E2 -10082.888} C_VEL
LIN {X 0,Y 418.437,Z 146.359,A -85,B 0,C 180,E1 -10086.752,E2 -10086.752} C_VEL
LIN {X 0,Y 418.315,Z 146.379,A -85,B 0,C 180,E1 -10089.672,E2 -10089.672} C_VEL
LIN {X 0,Y 418.336,Z 146.372,A -85,B 0,C 180,E1 -10092.996,E2 -10092.996} C_VEL
LIN {X 0,Y 418.253,Z 146.382,A -85,B 0,C 180,E1 -10096.709,E2 -10096.709} C_VEL
LIN {X 0,Y 418.238,Z 146.387,A -85,B 0,C 180,E1 -10099.778,E2 -10099.778} C_VEL
LIN {X 0,Y 418.222,Z 146.386,A -85,B 0,C 180,E1 -10102.737,E2 -10102.737} C_VEL
LIN {X 0,Y 418.215,Z 146.388,A -85,B 0,C 180,E1 -10105.908,E2 -10105.908} C_VEL
LIN {X 0,Y 418.252,Z 146.388,A -85,B 0,C 180,E1 -10109.163,E2 -10109.163} C_VEL
LIN {X 0,Y 418.246,Z 146.386,A -85,B 0,C 180,E1 -10112.842,E2 -10112.842} C_VEL
LIN {X 0,Y 418.241,Z 146.383,A -85,B 0,C 180,E1 -10116.238,E2 -10116.238} C_VEL
LIN {X 0,Y 418.208,Z 146.388,A -85,B 0,C 180,E1 -10119.687,E2 -10119.687} C_VEL
LIN {X 0,Y 418.207,Z 146.389,A -85,B 0,C 180,E1 -10122.318,E2 -10122.318} C_VEL
LIN {X 0,Y 418.235,Z 146.387,A -85,B 0,C 180,E1 -10125.109,E2 -10125.109} C_VEL
LIN {X 0,Y 418.218,Z 146.386,A -85,B 0,C 180,E1 -10127.764,E2 -10127.764} C_VEL
LIN {X 0,Y 418.238,Z 146.383,A -85,B 0,C 180,E1 -10131.557,E2 -10131.557} C_VEL
LIN {X 0,Y 418.251,Z 146.383,A -85,B 0,C 180,E1 -10135.158,E2 -10135.158} C_VEL
LIN {X 0,Y 418.244,Z 146.383,A -85,B 0,C 180,E1 -10137.472,E2 -10137.472} C_VEL
LIN {X 0,Y 418.263,Z 146.384,A -85,B 0,C 180,E1 -10140.897,E2 -10140.897} C_VEL
LIN {X 0,Y 418.311,Z 146.473,A -85,B 0,C 180,E1 -10142.278,E2 -10142.278} C_VEL
